  STRUCT
   STAT0 : ARRAY  [0 .. 255 ] OF //Temporary placeholder variable
   WORD  := W#16#0;
  END_STRUCT ;
BEGIN
   STAT0[0] := W#16#0;
   STAT0[1] := W#16#0;
   STAT0[2] := W#16#0;
   STAT0[3] := W#16#0;
   STAT0[4] := W#16#0;
   STAT0[5] := W#16#0;
   STAT0[6] := W#16#0;
   STAT0[7] := W#16#0;
   STAT0[8] := W#16#0;
   STAT0[9] := W#16#0;
   STAT0[10] := W#16#0;
   STAT0[11] := W#16#0;
   STAT0[12] := W#16#0;
   STAT0[13] := W#16#0;
   STAT0[14] := W#16#0;
   STAT0[15] := W#16#0;
   STAT0[16] := W#16#0;
   STAT0[17] := W#16#0;
   STAT0[18] := W#16#0;
   STAT0[19] := W#16#0;
   STAT0[20] := W#16#0;
   STAT0[21] := W#16#0;
   STAT0[22] := W#16#0;
   STAT0[23] := W#16#0;
   STAT0[24] := W#16#0;
   STAT0[25] := W#16#0;
   STAT0[26] := W#16#0;
   STAT0[27] := W#16#0;
   STAT0[28] := W#16#0;
   STAT0[29] := W#16#0;
   STAT0[30] := W#16#0;
   STAT0[31] := W#16#0;
   STAT0[32] := W#16#0;
   STAT0[33] := W#16#0;
   STAT0[34] := W#16#0;
   STAT0[35] := W#16#0;
   STAT0[36] := W#16#0;
   STAT0[37] := W#16#0;
   STAT0[38] := W#16#0;
   STAT0[39] := W#16#0;
   STAT0[40] := W#16#0;
   STAT0[41] := W#16#0;
   STAT0[42] := W#16#0;
   STAT0[43] := W#16#0;
   STAT0[44] := W#16#0;
   STAT0[45] := W#16#0;
   STAT0[46] := W#16#0;
   STAT0[47] := W#16#0;
   STAT0[48] := W#16#0;
   STAT0[49] := W#16#0;
   STAT0[50] := W#16#0;
   STAT0[51] := W#16#0;
   STAT0[52] := W#16#0;
   STAT0[53] := W#16#0;
   STAT0[54] := W#16#0;
   STAT0[55] := W#16#0;
   STAT0[56] := W#16#0;
   STAT0[57] := W#16#0;
   STAT0[58] := W#16#0;
   STAT0[59] := W#16#0;
   STAT0[60] := W#16#0;
   STAT0[61] := W#16#0;
   STAT0[62] := W#16#0;
   STAT0[63] := W#16#0;
   STAT0[64] := W#16#0;
   STAT0[65] := W#16#0;
   STAT0[66] := W#16#0;
   STAT0[67] := W#16#0;
   STAT0[68] := W#16#0;
   STAT0[69] := W#16#0;
   STAT0[70] := W#16#0;
   STAT0[71] := W#16#0;
   STAT0[72] := W#16#0;
   STAT0[73] := W#16#0;
   STAT0[74] := W#16#0;
   STAT0[75] := W#16#0;
   STAT0[76] := W#16#0;
   STAT0[77] := W#16#0;
   STAT0[78] := W#16#0;
   STAT0[79] := W#16#0;
   STAT0[80] := W#16#0;
   STAT0[81] := W#16#0;
   STAT0[82] := W#16#0;
   STAT0[83] := W#16#0;
   STAT0[84] := W#16#0;
   STAT0[85] := W#16#0;
   STAT0[86] := W#16#0;
   STAT0[87] := W#16#0;
   STAT0[88] := W#16#0;
   STAT0[89] := W#16#0;
   STAT0[90] := W#16#0;
   STAT0[91] := W#16#0;
   STAT0[92] := W#16#0;
   STAT0[93] := W#16#0;
   STAT0[94] := W#16#0;
   STAT0[95] := W#16#0;
   STAT0[96] := W#16#0;
   STAT0[97] := W#16#0;
   STAT0[98] := W#16#0;
   STAT0[99] := W#16#0;
   STAT0[100] := W#16#0;
   STAT0[101] := W#16#0;
   STAT0[102] := W#16#0;
   STAT0[103] := W#16#0;
   STAT0[104] := W#16#0;
   STAT0[105] := W#16#0;
   STAT0[106] := W#16#0;
   STAT0[107] := W#16#0;
   STAT0[108] := W#16#0;
   STAT0[109] := W#16#0;
   STAT0[110] := W#16#0;
   STAT0[111] := W#16#0;
   STAT0[112] := W#16#0;
   STAT0[113] := W#16#0;
   STAT0[114] := W#16#0;
   STAT0[115] := W#16#0;
   STAT0[116] := W#16#0;
   STAT0[117] := W#16#0;
   STAT0[118] := W#16#0;
   STAT0[119] := W#16#0;
   STAT0[120] := W#16#0;
   STAT0[121] := W#16#0;
   STAT0[122] := W#16#0;
   STAT0[123] := W#16#0;
   STAT0[124] := W#16#0;
   STAT0[125] := W#16#0;
   STAT0[126] := W#16#0;
   STAT0[127] := W#16#0;
   STAT0[128] := W#16#0;
   STAT0[129] := W#16#0;
   STAT0[130] := W#16#0;
   STAT0[131] := W#16#0;
   STAT0[132] := W#16#0;
   STAT0[133] := W#16#0;
   STAT0[134] := W#16#0;
   STAT0[135] := W#16#0;
   STAT0[136] := W#16#0;
   STAT0[137] := W#16#0;
   STAT0[138] := W#16#0;
   STAT0[139] := W#16#0;
   STAT0[140] := W#16#0;
   STAT0[141] := W#16#0;
   STAT0[142] := W#16#0;
   STAT0[143] := W#16#0;
   STAT0[144] := W#16#0;
   STAT0[145] := W#16#0;
   STAT0[146] := W#16#0;
   STAT0[147] := W#16#0;
   STAT0[148] := W#16#0;
   STAT0[149] := W#16#0;
   STAT0[150] := W#16#0;
   STAT0[151] := W#16#0;
   STAT0[152] := W#16#0;
   STAT0[153] := W#16#0;
   STAT0[154] := W#16#0;
   STAT0[155] := W#16#0;
   STAT0[156] := W#16#0;
   STAT0[157] := W#16#0;
   STAT0[158] := W#16#0;
   STAT0[159] := W#16#0;
   STAT0[160] := W#16#0;
   STAT0[161] := W#16#0;
   STAT0[162] := W#16#0;
   STAT0[163] := W#16#0;
   STAT0[164] := W#16#0;
   STAT0[165] := W#16#0;
   STAT0[166] := W#16#0;
   STAT0[167] := W#16#0;
   STAT0[168] := W#16#0;
   STAT0[169] := W#16#0;
   STAT0[170] := W#16#0;
   STAT0[171] := W#16#0;
   STAT0[172] := W#16#0;
   STAT0[173] := W#16#0;
   STAT0[174] := W#16#0;
   STAT0[175] := W#16#0;
   STAT0[176] := W#16#0;
   STAT0[177] := W#16#0;
   STAT0[178] := W#16#0;
   STAT0[179] := W#16#0;
   STAT0[180] := W#16#0;
   STAT0[181] := W#16#0;
   STAT0[182] := W#16#0;
   STAT0[183] := W#16#0;
   STAT0[184] := W#16#0;
   STAT0[185] := W#16#0;
   STAT0[186] := W#16#0;
   STAT0[187] := W#16#0;
   STAT0[188] := W#16#0;
   STAT0[189] := W#16#0;
   STAT0[190] := W#16#0;
   STAT0[191] := W#16#0;
   STAT0[192] := W#16#0;
   STAT0[193] := W#16#0;
   STAT0[194] := W#16#0;
   STAT0[195] := W#16#0;
   STAT0[196] := W#16#0;
   STAT0[197] := W#16#0;
   STAT0[198] := W#16#0;
   STAT0[199] := W#16#0;
   STAT0[200] := W#16#0;
   STAT0[201] := W#16#0;
   STAT0[202] := W#16#0;
   STAT0[203] := W#16#0;
   STAT0[204] := W#16#0;
   STAT0[205] := W#16#0;
   STAT0[206] := W#16#0;
   STAT0[207] := W#16#0;
   STAT0[208] := W#16#0;
   STAT0[209] := W#16#0;
   STAT0[210] := W#16#0;
   STAT0[211] := W#16#0;
   STAT0[212] := W#16#0;
   STAT0[213] := W#16#0;
   STAT0[214] := W#16#0;
   STAT0[215] := W#16#0;
   STAT0[216] := W#16#0;
   STAT0[217] := W#16#0;
   STAT0[218] := W#16#0;
   STAT0[219] := W#16#0;
   STAT0[220] := W#16#0;
   STAT0[221] := W#16#0;
   STAT0[222] := W#16#0;
   STAT0[223] := W#16#0;
   STAT0[224] := W#16#0;
   STAT0[225] := W#16#0;
   STAT0[226] := W#16#0;
   STAT0[227] := W#16#0;
   STAT0[228] := W#16#0;
   STAT0[229] := W#16#0;
   STAT0[230] := W#16#0;
   STAT0[231] := W#16#0;
   STAT0[232] := W#16#0;
   STAT0[233] := W#16#0;
   STAT0[234] := W#16#0;
   STAT0[235] := W#16#0;
   STAT0[236] := W#16#0;
   STAT0[237] := W#16#0;
   STAT0[238] := W#16#0;
   STAT0[239] := W#16#0;
   STAT0[240] := W#16#0;
   STAT0[241] := W#16#0;
   STAT0[242] := W#16#0;
   STAT0[243] := W#16#0;
   STAT0[244] := W#16#0;
   STAT0[245] := W#16#0;
   STAT0[246] := W#16#0;
   STAT0[247] := W#16#0;
   STAT0[248] := W#16#0;
   STAT0[249] := W#16#0;
   STAT0[250] := W#16#0;
   STAT0[251] := W#16#0;
   STAT0[252] := W#16#0;
   STAT0[253] := W#16#0;
   STAT0[254] := W#16#0;
   STAT0[255] := W#16#0;
END_DATA_BLOCK

DATA_BLOCK DB 325
TITLE =
VERSION : 0.1


  STRUCT
   DP_DIAG1 : ARRAY  [1 .. 100 ] OF BYTE ;
   DP_DIAG2 : ARRAY  [1 .. 100 ] OF BYTE ;
   DP_DIAG3 : ARRAY  [1 .. 100 ] OF BYTE ;
   DP_DIAG4 : ARRAY  [1 .. 100 ] OF BYTE ;
   DP_DIAG5 : ARRAY  [1 .. 100 ] OF BYTE ;
   DP_DIAG6 : ARRAY  [1 .. 100 ] OF BYTE ;
   DP_DIAG7 : ARRAY  [1 .. 100 ] OF BYTE ;
   DP_DIAG8 : ARRAY  [1 .. 100 ] OF BYTE ;
   DP_DIAG9 : ARRAY  [1 .. 100 ] OF BYTE ;
   DP_DIAG10 : ARRAY  [1 .. 100 ] OF BYTE ;
  END_STRUCT ;
BEGIN
   DP_DIAG1[1] := B#16#0;
   DP_DIAG1[2] := B#16#0;
   DP_DIAG1[3] := B#16#0;
   DP_DIAG1[4] := B#16#0;
   DP_DIAG1[5] := B#16#0;
   DP_DIAG1[6] := B#16#0;
   DP_DIAG1[7] := B#16#0;
   DP_DIAG1[8] := B#16#0;
   DP_DIAG1[9] := B#16#0;
   DP_DIAG1[10] := B#16#0;
   DP_DIAG1[11] := B#16#0;
   DP_DIAG1[12] := B#16#0;
   DP_DIAG1[13] := B#16#0;
   DP_DIAG1[14] := B#16#0;
   DP_DIAG1[15] := B#16#0;
   DP_DIAG1[16] := B#16#0;
   DP_DIAG1[17] := B#16#0;
   DP_DIAG1[18] := B#16#0;
   DP_DIAG1[19] := B#16#0;
   DP_DIAG1[20] := B#16#0;
   DP_DIAG1[21] := B#16#0;
   DP_DIAG1[22] := B#16#0;
   DP_DIAG1[23] := B#16#0;
   DP_DIAG1[24] := B#16#0;
   DP_DIAG1[25] := B#16#0;
   DP_DIAG1[26] := B#16#0;
   DP_DIAG1[27] := B#16#0;
   DP_DIAG1[28] := B#16#0;
   DP_DIAG1[29] := B#16#0;
   DP_DIAG1[30] := B#16#0;
   DP_DIAG1[31] := B#16#0;
   DP_DIAG1[32] := B#16#0;
   DP_DIAG1[33] := B#16#0;
   DP_DIAG1[34] := B#16#0;
   DP_DIAG1[35] := B#16#0;
   DP_DIAG1[36] := B#16#0;
   DP_DIAG1[37] := B#16#0;
   DP_DIAG1[38] := B#16#0;
   DP_DIAG1[39] := B#16#0;
   DP_DIAG1[40] := B#16#0;
   DP_DIAG1[41] := B#16#0;
   DP_DIAG1[42] := B#16#0;
   DP_DIAG1[43] := B#16#0;
   DP_DIAG1[44] := B#16#0;
   DP_DIAG1[45] := B#16#0;
   DP_DIAG1[46] := B#16#0;
   DP_DIAG1[47] := B#16#0;
   DP_DIAG1[48] := B#16#0;
   DP_DIAG1[49] := B#16#0;
   DP_DIAG1[50] := B#16#0;
   DP_DIAG1[51] := B#16#0;
   DP_DIAG1[52] := B#16#0;
   DP_DIAG1[53] := B#16#0;
   DP_DIAG1[54] := B#16#0;
   DP_DIAG1[55] := B#16#0;
   DP_DIAG1[56] := B#16#0;
   DP_DIAG1[57] := B#16#0;
   DP_DIAG1[58] := B#16#0;
   DP_DIAG1[59] := B#16#0;
   DP_DIAG1[60] := B#16#0;
   DP_DIAG1[61] := B#16#0;
   DP_DIAG1[62] := B#16#0;
   DP_DIAG1[63] := B#16#0;
   DP_DIAG1[64] := B#16#0;
   DP_DIAG1[65] := B#16#0;
   DP_DIAG1[66] := B#16#0;
   DP_DIAG1[67] := B#16#0;
   DP_DIAG1[68] := B#16#0;
   DP_DIAG1[69] := B#16#0;
   DP_DIAG1[70] := B#16#0;
   DP_DIAG1[71] := B#16#0;
   DP_DIAG1[72] := B#16#0;
   DP_DIAG1[73] := B#16#0;
   DP_DIAG1[74] := B#16#0;
   DP_DIAG1[75] := B#16#0;
   DP_DIAG1[76] := B#16#0;
   DP_DIAG1[77] := B#16#0;
   DP_DIAG1[78] := B#16#0;
   DP_DIAG1[79] := B#16#0;
   DP_DIAG1[80] := B#16#0;
   DP_DIAG1[81] := B#16#0;
   DP_DIAG1[82] := B#16#0;
   DP_DIAG1[83] := B#16#0;
   DP_DIAG1[84] := B#16#0;
   DP_DIAG1[85] := B#16#0;
   DP_DIAG1[86] := B#16#0;
   DP_DIAG1[87] := B#16#0;
   DP_DIAG1[88] := B#16#0;
   DP_DIAG1[89] := B#16#0;
   DP_DIAG1[90] := B#16#0;
   DP_DIAG1[91] := B#16#0;
   DP_DIAG1[92] := B#16#0;
   DP_DIAG1[93] := B#16#0;
   DP_DIAG1[94] := B#16#0;
   DP_DIAG1[95] := B#16#0;
   DP_DIAG1[96] := B#16#0;
   DP_DIAG1[97] := B#16#0;
   DP_DIAG1[98] := B#16#0;
   DP_DIAG1[99] := B#16#0;
   DP_DIAG1[100] := B#16#0;
   DP_DIAG2[1] := B#16#0;
   DP_DIAG2[2] := B#16#0;
   DP_DIAG2[3] := B#16#0;
   DP_DIAG2[4] := B#16#0;
   DP_DIAG2[5] := B#16#0;
   DP_DIAG2[6] := B#16#0;
   DP_DIAG2[7] := B#16#0;
   DP_DIAG2[8] := B#16#0;
   DP_DIAG2[9] := B#16#0;
   DP_DIAG2[10] := B#16#0;
   DP_DIAG2[11] := B#16#0;
   DP_DIAG2[12] := B#16#0;
   DP_DIAG2[13] := B#16#0;
   DP_DIAG2[14] := B#16#0;
   DP_DIAG2[15] := B#16#0;
   DP_DIAG2[16] := B#16#0;
   DP_DIAG2[17] := B#16#0;
   DP_DIAG2[18] := B#16#0;
   DP_DIAG2[19] := B#16#0;
   DP_DIAG2[20] := B#16#0;
   DP_DIAG2[21] := B#16#0;
   DP_DIAG2[22] := B#16#0;
   DP_DIAG2[23] := B#16#0;
   DP_DIAG2[24] := B#16#0;
   DP_DIAG2[25] := B#16#0;
   DP_DIAG2[26] := B#16#0;
   DP_DIAG2[27] := B#16#0;
   DP_DIAG2[28] := B#16#0;
   DP_DIAG2[29] := B#16#0;
   DP_DIAG2[30] := B#16#0;
   DP_DIAG2[31] := B#16#0;
   DP_DIAG2[32] := B#16#0;
   DP_DIAG2[33] := B#16#0;
   DP_DIAG2[34] := B#16#0;
   DP_DIAG2[35] := B#16#0;
   DP_DIAG2[36] := B#16#0;
   DP_DIAG2[37] := B#16#0;
   DP_DIAG2[38] := B#16#0;
   DP_DIAG2[39] := B#16#0;
   DP_DIAG2[40] := B#16#0;
   DP_DIAG2[41] := B#16#0;
   DP_DIAG2[42] := B#16#0;
   DP_DIAG2[43] := B#16#0;
   DP_DIAG2[44] := B#16#0;
   DP_DIAG2[45] := B#16#0;
   DP_DIAG2[46] := B#16#0;
   DP_DIAG2[47] := B#16#0;
   DP_DIAG2[48] := B#16#0;
   DP_DIAG2[49] := B#16#0;
   DP_DIAG2[50] := B#16#0;
   DP_DIAG2[51] := B#16#0;
   DP_DIAG2[52] := B#16#0;
   DP_DIAG2[53] := B#16#0;
   DP_DIAG2[54] := B#16#0;
   DP_DIAG2[55] := B#16#0;
   DP_DIAG2[56] := B#16#0;
   DP_DIAG2[57] := B#16#0;
   DP_DIAG2[58] := B#16#0;
   DP_DIAG2[59] := B#16#0;
   DP_DIAG2[60] := B#16#0;
   DP_DIAG2[61] := B#16#0;
   DP_DIAG2[62] := B#16#0;
   DP_DIAG2[63] := B#16#0;
   DP_DIAG2[64] := B#16#0;
   DP_DIAG2[65] := B#16#0;
   DP_DIAG2[66] := B#16#0;
   DP_DIAG2[67] := B#16#0;
   DP_DIAG2[68] := B#16#0;
   DP_DIAG2[69] := B#16#0;
   DP_DIAG2[70] := B#16#0;
   DP_DIAG2[71] := B#16#0;
   DP_DIAG2[72] := B#16#0;
   DP_DIAG2[73] := B#16#0;
   DP_DIAG2[74] := B#16#0;
   DP_DIAG2[75] := B#16#0;
   DP_DIAG2[76] := B#16#0;
   DP_DIAG2[77] := B#16#0;
   DP_DIAG2[78] := B#16#0;
   DP_DIAG2[79] := B#16#0;
   DP_DIAG2[80] := B#16#0;
   DP_DIAG2[81] := B#16#0;
   DP_DIAG2[82] := B#16#0;
   DP_DIAG2[83] := B#16#0;
   DP_DIAG2[84] := B#16#0;
   DP_DIAG2[85] := B#16#0;
   DP_DIAG2[86] := B#16#0;
   DP_DIAG2[87] := B#16#0;
   DP_DIAG2[88] := B#16#0;
   DP_DIAG2[89] := B#16#0;
   DP_DIAG2[90] := B#16#0;
   DP_DIAG2[91] := B#16#0;
   DP_DIAG2[92] := B#16#0;
   DP_DIAG2[93] := B#16#0;
   DP_DIAG2[94] := B#16#0;
   DP_DIAG2[95] := B#16#0;
   DP_DIAG2[96] := B#16#0;
   DP_DIAG2[97] := B#16#0;
   DP_DIAG2[98] := B#16#0;
   DP_DIAG2[99] := B#16#0;
   DP_DIAG2[100] := B#16#0;
   DP_DIAG3[1] := B#16#0;
   DP_DIAG3[2] := B#16#0;
   DP_DIAG3[3] := B#16#0;
   DP_DIAG3[4] := B#16#0;
   DP_DIAG3[5] := B#16#0;
   DP_DIAG3[6] := B#16#0;
   DP_DIAG3[7] := B#16#0;
   DP_DIAG3[8] := B#16#0;
   DP_DIAG3[9] := B#16#0;
   DP_DIAG3[10] := B#16#0;
   DP_DIAG3[11] := B#16#0;
   DP_DIAG3[12] := B#16#0;
   DP_DIAG3[13] := B#16#0;
   DP_DIAG3[14] := B#16#0;
   DP_DIAG3[15] := B#16#0;
   DP_DIAG3[16] := B#16#0;
   DP_DIAG3[17] := B#16#0;
   DP_DIAG3[18] := B#16#0;
   DP_DIAG3[19] := B#16#0;
   DP_DIAG3[20] := B#16#0;
   DP_DIAG3[21] := B#16#0;
   DP_DIAG3[22] := B#16#0;
   DP_DIAG3[23] := B#16#0;
   DP_DIAG3[24] := B#16#0;
   DP_DIAG3[25] := B#16#0;
   DP_DIAG3[26] := B#16#0;
   DP_DIAG3[27] := B#16#0;
   DP_DIAG3[28] := B#16#0;
   DP_DIAG3[29] := B#16#0;
   DP_DIAG3[30] := B#16#0;
   DP_DIAG3[31] := B#16#0;
   DP_DIAG3[32] := B#16#0;
   DP_DIAG3[33] := B#16#0;
   DP_DIAG3[34] := B#16#0;
   DP_DIAG3[35] := B#16#0;
   DP_DIAG3[36] := B#16#0;
   DP_DIAG3[37] := B#16#0;
   DP_DIAG3[38] := B#16#0;
   DP_DIAG3[39] := B#16#0;
   DP_DIAG3[40] := B#16#0;
   DP_DIAG3[41] := B#16#0;
   DP_DIAG3[42] := B#16#0;
   DP_DIAG3[43] := B#16#0;
   DP_DIAG3[44] := B#16#0;
   DP_DIAG3[45] := B#16#0;
   DP_DIAG3[46] := B#16#0;
   DP_DIAG3[47] := B#16#0;
   DP_DIAG3[48] := B#16#0;
   DP_DIAG3[49] := B#16#0;
   DP_DIAG3[50] := B#16#0;
   DP_DIAG3[51] := B#16#0;
   DP_DIAG3[52] := B#16#0;
   DP_DIAG3[53] := B#16#0;
   DP_DIAG3[54] := B#16#0;
   DP_DIAG3[55] := B#16#0;
   DP_DIAG3[56] := B#16#0;
   DP_DIAG3[57] := B#16#0;
   DP_DIAG3[58] := B#16#0;
   DP_DIAG3[59] := B#16#0;
   DP_DIAG3[60] := B#16#0;
   DP_DIAG3[61] := B#16#0;
   DP_DIAG3[62] := B#16#0;
   DP_DIAG3[63] := B#16#0;
   DP_DIAG3[64] := B#16#0;
   DP_DIAG3[65] := B#16#0;
   DP_DIAG3[66] := B#16#0;
   DP_DIAG3[67] := B#16#0;
   DP_DIAG3[68] := B#16#0;
   DP_DIAG3[69] := B#16#0;
   DP_DIAG3[70] := B#16#0;
   DP_DIAG3[71] := B#16#0;
   DP_DIAG3[72] := B#16#0;
   DP_DIAG3[73] := B#16#0;
   DP_DIAG3[74] := B#16#0;
   DP_DIAG3[75] := B#16#0;
   DP_DIAG3[76] := B#16#0;
   DP_DIAG3[77] := B#16#0;
   DP_DIAG3[78] := B#16#0;
   DP_DIAG3[79] := B#16#0;
   DP_DIAG3[80] := B#16#0;
   DP_DIAG3[81] := B#16#0;
   DP_DIAG3[82] := B#16#0;
   DP_DIAG3[83] := B#16#0;
   DP_DIAG3[84] := B#16#0;
   DP_DIAG3[85] := B#16#0;
   DP_DIAG3[86] := B#16#0;
   DP_DIAG3[87] := B#16#0;
   DP_DIAG3[88] := B#16#0;
   DP_DIAG3[89] := B#16#0;
   DP_DIAG3[90] := B#16#0;
   DP_DIAG3[91] := B#16#0;
   DP_DIAG3[92] := B#16#0;
   DP_DIAG3[93] := B#16#0;
   DP_DIAG3[94] := B#16#0;
   DP_DIAG3[95] := B#16#0;
   DP_DIAG3[96] := B#16#0;
   DP_DIAG3[97] := B#16#0;
   DP_DIAG3[98] := B#16#0;
   DP_DIAG3[99] := B#16#0;
   DP_DIAG3[100] := B#16#0;
   DP_DIAG4[1] := B#16#0;
   DP_DIAG4[2] := B#16#0;
   DP_DIAG4[3] := B#16#0;
   DP_DIAG4[4] := B#16#0;
   DP_DIAG4[5] := B#16#0;
   DP_DIAG4[6] := B#16#0;
   DP_DIAG4[7] := B#16#0;
   DP_DIAG4[8] := B#16#0;
   DP_DIAG4[9] := B#16#0;
   DP_DIAG4[10] := B#16#0;
   DP_DIAG4[11] := B#16#0;
   DP_DIAG4[12] := B#16#0;
   DP_DIAG4[13] := B#16#0;
   DP_DIAG4[14] := B#16#0;
   DP_DIAG4[15] := B#16#0;
   DP_DIAG4[16] := B#16#0;
   DP_DIAG4[17] := B#16#0;
   DP_DIAG4[18] := B#16#0;
   DP_DIAG4[19] := B#16#0;
   DP_DIAG4[20] := B#16#0;
   DP_DIAG4[21] := B#16#0;
   DP_DIAG4[22] := B#16#0;
   DP_DIAG4[23] := B#16#0;
   DP_DIAG4[24] := B#16#0;
   DP_DIAG4[25] := B#16#0;
   DP_DIAG4[26] := B#16#0;
   DP_DIAG4[27] := B#16#0;
   DP_DIAG4[28] := B#16#0;
   DP_DIAG4[29] := B#16#0;
   DP_DIAG4[30] := B#16#0;
   DP_DIAG4[31] := B#16#0;
   DP_DIAG4[32] := B#16#0;
   DP_DIAG4[33] := B#16#0;
   DP_DIAG4[34] := B#16#0;
   DP_DIAG4[35] := B#16#0;
   DP_DIAG4[36] := B#16#0;
   DP_DIAG4[37] := B#16#0;
   DP_DIAG4[38] := B#16#0;
   DP_DIAG4[39] := B#16#0;
   DP_DIAG4[40] := B#16#0;
   DP_DIAG4[41] := B#16#0;
   DP_DIAG4[42] := B#16#0;
   DP_DIAG4[43] := B#16#0;
   DP_DIAG4[44] := B#16#0;
   DP_DIAG4[45] := B#16#0;
   DP_DIAG4[46] := B#16#0;
   DP_DIAG4[47] := B#16#0;
   DP_DIAG4[48] := B#16#0;
   DP_DIAG4[49] := B#16#0;
   DP_DIAG4[50] := B#16#0;
   DP_DIAG4[51] := B#16#0;
   DP_DIAG4[52] := B#16#0;
   DP_DIAG4[53] := B#16#0;
   DP_DIAG4[54] := B#16#0;
   DP_DIAG4[55] := B#16#0;
   DP_DIAG4[56] := B#16#0;
   DP_DIAG4[57] := B#16#0;
   DP_DIAG4[58] := B#16#0;
   DP_DIAG4[59] := B#16#0;
   DP_DIAG4[60] := B#16#0;
   DP_DIAG4[61] := B#16#0;
   DP_DIAG4[62] := B#16#0;
   DP_DIAG4[63] := B#16#0;
   DP_DIAG4[64] := B#16#0;
   DP_DIAG4[65] := B#16#0;
   DP_DIAG4[66] := B#16#0;
   DP_DIAG4[67] := B#16#0;
   DP_DIAG4[68] := B#16#0;
   DP_DIAG4[69] := B#16#0;
   DP_DIAG4[70] := B#16#0;
   DP_DIAG4[71] := B#16#0;
   DP_DIAG4[72] := B#16#0;
   DP_DIAG4[73] := B#16#0;
   DP_DIAG4[74] := B#16#0;
   DP_DIAG4[75] := B#16#0;
   DP_DIAG4[76] := B#16#0;
   DP_DIAG4[77] := B#16#0;
   DP_DIAG4[78] := B#16#0;
   DP_DIAG4[79] := B#16#0;
   DP_DIAG4[80] := B#16#0;
   DP_DIAG4[81] := B#16#0;
   DP_DIAG4[82] := B#16#0;
   DP_DIAG4[83] := B#16#0;
   DP_DIAG4[84] := B#16#0;
   DP_DIAG4[85] := B#16#0;
   DP_DIAG4[86] := B#16#0;
   DP_DIAG4[87] := B#16#0;
   DP_DIAG4[88] := B#16#0;
   DP_DIAG4[89] := B#16#0;
   DP_DIAG4[90] := B#16#0;
   DP_DIAG4[91] := B#16#0;
   DP_DIAG4[92] := B#16#0;
   DP_DIAG4[93] := B#16#0;
   DP_DIAG4[94] := B#16#0;
   DP_DIAG4[95] := B#16#0;
   DP_DIAG4[96] := B#16#0;
   DP_DIAG4[97] := B#16#0;
   DP_DIAG4[98] := B#16#0;
   DP_DIAG4[99] := B#16#0;
   DP_DIAG4[100] := B#16#0;
   DP_DIAG5[1] := B#16#0;
   DP_DIAG5[2] := B#16#0;
   DP_DIAG5[3] := B#16#0;
   DP_DIAG5[4] := B#16#0;
   DP_DIAG5[5] := B#16#0;
   DP_DIAG5[6] := B#16#0;
   DP_DIAG5[7] := B#16#0;
   DP_DIAG5[8] := B#16#0;
   DP_DIAG5[9] := B#16#0;
   DP_DIAG5[10] := B#16#0;
   DP_DIAG5[11] := B#16#0;
   DP_DIAG5[12] := B#16#0;
   DP_DIAG5[13] := B#16#0;
   DP_DIAG5[14] := B#16#0;
   DP_DIAG5[15] := B#16#0;
   DP_DIAG5[16] := B#16#0;
   DP_DIAG5[17] := B#16#0;
   DP_DIAG5[18] := B#16#0;
   DP_DIAG5[19] := B#16#0;
   DP_DIAG5[20] := B#16#0;
   DP_DIAG5[21] := B#16#0;
   DP_DIAG5[22] := B#16#0;
   DP_DIAG5[23] := B#16#0;
   DP_DIAG5[24] := B#16#0;
   DP_DIAG5[25] := B#16#0;
   DP_DIAG5[26] := B#16#0;
   DP_DIAG5[27] := B#16#0;
   DP_DIAG5[28] := B#16#0;
   DP_DIAG5[29] := B#16#0;
   DP_DIAG5[30] := B#16#0;
   DP_DIAG5[31] := B#16#0;
   DP_DIAG5[32] := B#16#0;
   DP_DIAG5[33] := B#16#0;
   DP_DIAG5[34] := B#16#0;
   DP_DIAG5[35] := B#16#0;
   DP_DIAG5[36] := B#16#0;
   DP_DIAG5[37] := B#16#0;
   DP_DIAG5[38] := B#16#0;
   DP_DIAG5[39] := B#16#0;
   DP_DIAG5[40] := B#16#0;
   DP_DIAG5[41] := B#16#0;
   DP_DIAG5[42] := B#16#0;
   DP_DIAG5[43] := B#16#0;
   DP_DIAG5[44] := B#16#0;
   DP_DIAG5[45] := B#16#0;
   DP_DIAG5[46] := B#16#0;
   DP_DIAG5[47] := B#16#0;
   DP_DIAG5[48] := B#16#0;
   DP_DIAG5[49] := B#16#0;
   DP_DIAG5[50] := B#16#0;
   DP_DIAG5[51] := B#16#0;
   DP_DIAG5[52] := B#16#0;
   DP_DIAG5[53] := B#16#0;
   DP_DIAG5[54] := B#16#0;
   DP_DIAG5[55] := B#16#0;
   DP_DIAG5[56] := B#16#0;
   DP_DIAG5[57] := B#16#0;
   DP_DIAG5[58] := B#16#0;
   DP_DIAG5[59] := B#16#0;
   DP_DIAG5[60] := B#16#0;
   DP_DIAG5[61] := B#16#0;
   DP_DIAG5[62] := B#16#0;
   DP_DIAG5[63] := B#16#0;
   DP_DIAG5[64] := B#16#0;
   DP_DIAG5[65] := B#16#0;
   DP_DIAG5[66] := B#16#0;
   DP_DIAG5[67] := B#16#0;
   DP_DIAG5[68] := B#16#0;
   DP_DIAG5[69] := B#16#0;
   DP_DIAG5[70] := B#16#0;
   DP_DIAG5[71] := B#16#0;
   DP_DIAG5[72] := B#16#0;
   DP_DIAG5[73] := B#16#0;
   DP_DIAG5[74] := B#16#0;
   DP_DIAG5[75] := B#16#0;
   DP_DIAG5[76] := B#16#0;
   DP_DIAG5[77] := B#16#0;
   DP_DIAG5[78] := B#16#0;
   DP_DIAG5[79] := B#16#0;
   DP_DIAG5[80] := B#16#0;
   DP_DIAG5[81] := B#16#0;
   DP_DIAG5[82] := B#16#0;
   DP_DIAG5[83] := B#16#0;
   DP_DIAG5[84] := B#16#0;
   DP_DIAG5[85] := B#16#0;
   DP_DIAG5[86] := B#16#0;
   DP_DIAG5[87] := B#16#0;
   DP_DIAG5[88] := B#16#0;
   DP_DIAG5[89] := B#16#0;
   DP_DIAG5[90] := B#16#0;
   DP_DIAG5[91] := B#16#0;
   DP_DIAG5[92] := B#16#0;
   DP_DIAG5[93] := B#16#0;
   DP_DIAG5[94] := B#16#0;
   DP_DIAG5[95] := B#16#0;
   DP_DIAG5[96] := B#16#0;
   DP_DIAG5[97] := B#16#0;
   DP_DIAG5[98] := B#16#0;
   DP_DIAG5[99] := B#16#0;
   DP_DIAG5[100] := B#16#0;
   DP_DIAG6[1] := B#16#0;
   DP_DIAG6[2] := B#16#0;
   DP_DIAG6[3] := B#16#0;
   DP_DIAG6[4] := B#16#0;
   DP_DIAG6[5] := B#16#0;
   DP_DIAG6[6] := B#16#0;
   DP_DIAG6[7] := B#16#0;
   DP_DIAG6[8] := B#16#0;
   DP_DIAG6[9] := B#16#0;
   DP_DIAG6[10] := B#16#0;
   DP_DIAG6[11] := B#16#0;
   DP_DIAG6[12] := B#16#0;
   DP_DIAG6[13] := B#16#0;
   DP_DIAG6[14] := B#16#0;
   DP_DIAG6[15] := B#16#0;
   DP_DIAG6[16] := B#16#0;
   DP_DIAG6[17] := B#16#0;
   DP_DIAG6[18] := B#16#0;
   DP_DIAG6[19] := B#16#0;
   DP_DIAG6[20] := B#16#0;
   DP_DIAG6[21] := B#16#0;
   DP_DIAG6[22] := B#16#0;
   DP_DIAG6[23] := B#16#0;
   DP_DIAG6[24] := B#16#0;
   DP_DIAG6[25] := B#16#0;
   DP_DIAG6[26] := B#16#0;
   DP_DIAG6[27] := B#16#0;
   DP_DIAG6[28] := B#16#0;
   DP_DIAG6[29] := B#16#0;
   DP_DIAG6[30] := B#16#0;
   DP_DIAG6[31] := B#16#0;
   DP_DIAG6[32] := B#16#0;
   DP_DIAG6[33] := B#16#0;
   DP_DIAG6[34] := B#16#0;
   DP_DIAG6[35] := B#16#0;
   DP_DIAG6[36] := B#16#0;
   DP_DIAG6[37] := B#16#0;
   DP_DIAG6[38] := B#16#0;
   DP_DIAG6[39] := B#16#0;
   DP_DIAG6[40] := B#16#0;
   DP_DIAG6[41] := B#16#0;
   DP_DIAG6[42] := B#16#0;
   DP_DIAG6[43] := B#16#0;
   DP_DIAG6[44] := B#16#0;
   DP_DIAG6[45] := B#16#0;
   DP_DIAG6[46] := B#16#0;
   DP_DIAG6[47] := B#16#0;
   DP_DIAG6[48] := B#16#0;
   DP_DIAG6[49] := B#16#0;
   DP_DIAG6[50] := B#16#0;
   DP_DIAG6[51] := B#16#0;
   DP_DIAG6[52] := B#16#0;
   DP_DIAG6[53] := B#16#0;
   DP_DIAG6[54] := B#16#0;
   DP_DIAG6[55] := B#16#0;
   DP_DIAG6[56] := B#16#0;
   DP_DIAG6[57] := B#16#0;
   DP_DIAG6[58] := B#16#0;
   DP_DIAG6[59] := B#16#0;
   DP_DIAG6[60] := B#16#0;
   DP_DIAG6[61] := B#16#0;
   DP_DIAG6[62] := B#16#0;
   DP_DIAG6[63] := B#16#0;
   DP_DIAG6[64] := B#16#0;
   DP_DIAG6[65] := B#16#0;
   DP_DIAG6[66] := B#16#0;
   DP_DIAG6[67] := B#16#0;
   DP_DIAG6[68] := B#16#0;
   DP_DIAG6[69] := B#16#0;
   DP_DIAG6[70] := B#16#0;
   DP_DIAG6[71] := B#16#0;
   DP_DIAG6[72] := B#16#0;
   DP_DIAG6[73] := B#16#0;
   DP_DIAG6[74] := B#16#0;
   DP_DIAG6[75] := B#16#0;
   DP_DIAG6[76] := B#16#0;
   DP_DIAG6[77] := B#16#0;
   DP_DIAG6[78] := B#16#0;
   DP_DIAG6[79] := B#16#0;
   DP_DIAG6[80] := B#16#0;
   DP_DIAG6[81] := B#16#0;
   DP_DIAG6[82] := B#16#0;
   DP_DIAG6[83] := B#16#0;
   DP_DIAG6[84] := B#16#0;
   DP_DIAG6[85] := B#16#0;
   DP_DIAG6[86] := B#16#0;
   DP_DIAG6[87] := B#16#0;
   DP_DIAG6[88] := B#16#0;
   DP_DIAG6[89] := B#16#0;
   DP_DIAG6[90] := B#16#0;
   DP_DIAG6[91] := B#16#0;
   DP_DIAG6[92] := B#16#0;
   DP_DIAG6[93] := B#16#0;
   DP_DIAG6[94] := B#16#0;
   DP_DIAG6[95] := B#16#0;
   DP_DIAG6[96] := B#16#0;
   DP_DIAG6[97] := B#16#0;
   DP_DIAG6[98] := B#16#0;
   DP_DIAG6[99] := B#16#0;
   DP_DIAG6[100] := B#16#0;
   DP_DIAG7[1] := B#16#0;
   DP_DIAG7[2] := B#16#0;
   DP_DIAG7[3] := B#16#0;
   DP_DIAG7[4] := B#16#0;
   DP_DIAG7[5] := B#16#0;
   DP_DIAG7[6] := B#16#0;
   DP_DIAG7[7] := B#16#0;
   DP_DIAG7[8] := B#16#0;
   DP_DIAG7[9] := B#16#0;
   DP_DIAG7[10] := B#16#0;
   DP_DIAG7[11] := B#16#0;
   DP_DIAG7[12] := B#16#0;
   DP_DIAG7[13] := B#16#0;
   DP_DIAG7[14] := B#16#0;
   DP_DIAG7[15] := B#16#0;
   DP_DIAG7[16] := B#16#0;
   DP_DIAG7[17] := B#16#0;
   DP_DIAG7[18] := B#16#0;
   DP_DIAG7[19] := B#16#0;
   DP_DIAG7[20] := B#16#0;
   DP_DIAG7[21] := B#16#0;
   DP_DIAG7[22] := B#16#0;
   DP_DIAG7[23] := B#16#0;
   DP_DIAG7[24] := B#16#0;
   DP_DIAG7[25] := B#16#0;
   DP_DIAG7[26] := B#16#0;
   DP_DIAG7[27] := B#16#0;
   DP_DIAG7[28] := B#16#0;
   DP_DIAG7[29] := B#16#0;
   DP_DIAG7[30] := B#16#0;
   DP_DIAG7[31] := B#16#0;
   DP_DIAG7[32] := B#16#0;
   DP_DIAG7[33] := B#16#0;
   DP_DIAG7[34] := B#16#0;
   DP_DIAG7[35] := B#16#0;
   DP_DIAG7[36] := B#16#0;
   DP_DIAG7[37] := B#16#0;
   DP_DIAG7[38] := B#16#0;
   DP_DIAG7[39] := B#16#0;
   DP_DIAG7[40] := B#16#0;
   DP_DIAG7[41] := B#16#0;
   DP_DIAG7[42] := B#16#0;
   DP_DIAG7[43] := B#16#0;
   DP_DIAG7[44] := B#16#0;
   DP_DIAG7[45] := B#16#0;
   DP_DIAG7[46] := B#16#0;
   DP_DIAG7[47] := B#16#0;
   DP_DIAG7[48] := B#16#0;
   DP_DIAG7[49] := B#16#0;
   DP_DIAG7[50] := B#16#0;
   DP_DIAG7[51] := B#16#0;
   DP_DIAG7[52] := B#16#0;
   DP_DIAG7[53] := B#16#0;
   DP_DIAG7[54] := B#16#0;
   DP_DIAG7[55] := B#16#0;
   DP_DIAG7[56] := B#16#0;
   DP_DIAG7[57] := B#16#0;
   DP_DIAG7[58] := B#16#0;
   DP_DIAG7[59] := B#16#0;
   DP_DIAG7[60] := B#16#0;
   DP_DIAG7[61] := B#16#0;
   DP_DIAG7[62] := B#16#0;
   DP_DIAG7[63] := B#16#0;
   DP_DIAG7[64] := B#16#0;
   DP_DIAG7[65] := B#16#0;
   DP_DIAG7[66] := B#16#0;
   DP_DIAG7[67] := B#16#0;
   DP_DIAG7[68] := B#16#0;
   DP_DIAG7[69] := B#16#0;
   DP_DIAG7[70] := B#16#0;
   DP_DIAG7[71] := B#16#0;
   DP_DIAG7[72] := B#16#0;
   DP_DIAG7[73] := B#16#0;
   DP_DIAG7[74] := B#16#0;
   DP_DIAG7[75] := B#16#0;
   DP_DIAG7[76] := B#16#0;
   DP_DIAG7[77] := B#16#0;
   DP_DIAG7[78] := B#16#0;
   DP_DIAG7[79] := B#16#0;
   DP_DIAG7[80] := B#16#0;
   DP_DIAG7[81] := B#16#0;
   DP_DIAG7[82] := B#16#0;
   DP_DIAG7[83] := B#16#0;
   DP_DIAG7[84] := B#16#0;
   DP_DIAG7[85] := B#16#0;
   DP_DIAG7[86] := B#16#0;
   DP_DIAG7[87] := B#16#0;
   DP_DIAG7[88] := B#16#0;
   DP_DIAG7[89] := B#16#0;
   DP_DIAG7[90] := B#16#0;
   DP_DIAG7[91] := B#16#0;
   DP_DIAG7[92] := B#16#0;
   DP_DIAG7[93] := B#16#0;
   DP_DIAG7[94] := B#16#0;
   DP_DIAG7[95] := B#16#0;
   DP_DIAG7[96] := B#16#0;
   DP_DIAG7[97] := B#16#0;
   DP_DIAG7[98] := B#16#0;
   DP_DIAG7[99] := B#16#0;
   DP_DIAG7[100] := B#16#0;
   DP_DIAG8[1] := B#16#0;
   DP_DIAG8[2] := B#16#0;
   DP_DIAG8[3] := B#16#0;
   DP_DIAG8[4] := B#16#0;
   DP_DIAG8[5] := B#16#0;
   DP_DIAG8[6] := B#16#0;
   DP_DIAG8[7] := B#16#0;
   DP_DIAG8[8] := B#16#0;
   DP_DIAG8[9] := B#16#0;
   DP_DIAG8[10] := B#16#0;
   DP_DIAG8[11] := B#16#0;
   DP_DIAG8[12] := B#16#0;
   DP_DIAG8[13] := B#16#0;
   DP_DIAG8[14] := B#16#0;
   DP_DIAG8[15] := B#16#0;
   DP_DIAG8[16] := B#16#0;
   DP_DIAG8[17] := B#16#0;
   DP_DIAG8[18] := B#16#0;
   DP_DIAG8[19] := B#16#0;
   DP_DIAG8[20] := B#16#0;
   DP_DIAG8[21] := B#16#0;
   DP_DIAG8[22] := B#16#0;
   DP_DIAG8[23] := B#16#0;
   DP_DIAG8[24] := B#16#0;
   DP_DIAG8[25] := B#16#0;
   DP_DIAG8[26] := B#16#0;
   DP_DIAG8[27] := B#16#0;
   DP_DIAG8[28] := B#16#0;
   DP_DIAG8[29] := B#16#0;
   DP_DIAG8[30] := B#16#0;
   DP_DIAG8[31] := B#16#0;
   DP_DIAG8[32] := B#16#0;
   DP_DIAG8[33] := B#16#0;
   DP_DIAG8[34] := B#16#0;
   DP_DIAG8[35] := B#16#0;
   DP_DIAG8[36] := B#16#0;
   DP_DIAG8[37] := B#16#0;
   DP_DIAG8[38] := B#16#0;
   DP_DIAG8[39] := B#16#0;
   DP_DIAG8[40] := B#16#0;
   DP_DIAG8[41] := B#16#0;
   DP_DIAG8[42] := B#16#0;
   DP_DIAG8[43] := B#16#0;
   DP_DIAG8[44] := B#16#0;
   DP_DIAG8[45] := B#16#0;
   DP_DIAG8[46] := B#16#0;
   DP_DIAG8[47] := B#16#0;
   DP_DIAG8[48] := B#16#0;
   DP_DIAG8[49] := B#16#0;
   DP_DIAG8[50] := B#16#0;
   DP_DIAG8[51] := B#16#0;
   DP_DIAG8[52] := B#16#0;
   DP_DIAG8[53] := B#16#0;
   DP_DIAG8[54] := B#16#0;
   DP_DIAG8[55] := B#16#0;
   DP_DIAG8[56] := B#16#0;
   DP_DIAG8[57] := B#16#0;
   DP_DIAG8[58] := B#16#0;
   DP_DIAG8[59] := B#16#0;
   DP_DIAG8[60] := B#16#0;
   DP_DIAG8[61] := B#16#0;
   DP_DIAG8[62] := B#16#0;
   DP_DIAG8[63] := B#16#0;
   DP_DIAG8[64] := B#16#0;
   DP_DIAG8[65] := B#16#0;
   DP_DIAG8[66] := B#16#0;
   DP_DIAG8[67] := B#16#0;
   DP_DIAG8[68] := B#16#0;
   DP_DIAG8[69] := B#16#0;
   DP_DIAG8[70] := B#16#0;
   DP_DIAG8[71] := B#16#0;
   DP_DIAG8[72] := B#16#0;
   DP_DIAG8[73] := B#16#0;
   DP_DIAG8[74] := B#16#0;
   DP_DIAG8[75] := B#16#0;
   DP_DIAG8[76] := B#16#0;
   DP_DIAG8[77] := B#16#0;
   DP_DIAG8[78] := B#16#0;
   DP_DIAG8[79] := B#16#0;
   DP_DIAG8[80] := B#16#0;
   DP_DIAG8[81] := B#16#0;
   DP_DIAG8[82] := B#16#0;
   DP_DIAG8[83] := B#16#0;
   DP_DIAG8[84] := B#16#0;
   DP_DIAG8[85] := B#16#0;
   DP_DIAG8[86] := B#16#0;
   DP_DIAG8[87] := B#16#0;
   DP_DIAG8[88] := B#16#0;
   DP_DIAG8[89] := B#16#0;
   DP_DIAG8[90] := B#16#0;
   DP_DIAG8[91] := B#16#0;
   DP_DIAG8[92] := B#16#0;
   DP_DIAG8[93] := B#16#0;
   DP_DIAG8[94] := B#16#0;
   DP_DIAG8[95] := B#16#0;
   DP_DIAG8[96] := B#16#0;
   DP_DIAG8[97] := B#16#0;
   DP_DIAG8[98] := B#16#0;
   DP_DIAG8[99] := B#16#0;
   DP_DIAG8[100] := B#16#0;
   DP_DIAG9[1] := B#16#0;
   DP_DIAG9[2] := B#16#0;
   DP_DIAG9[3] := B#16#0;
   DP_DIAG9[4] := B#16#0;
   DP_DIAG9[5] := B#16#0;
   DP_DIAG9[6] := B#16#0;
   DP_DIAG9[7] := B#16#0;
   DP_DIAG9[8] := B#16#0;
   DP_DIAG9[9] := B#16#0;
   DP_DIAG9[10] := B#16#0;
   DP_DIAG9[11] := B#16#0;
   DP_DIAG9[12] := B#16#0;
   DP_DIAG9[13] := B#16#0;
   DP_DIAG9[14] := B#16#0;
   DP_DIAG9[15] := B#16#0;
   DP_DIAG9[16] := B#16#0;
   DP_DIAG9[17] := B#16#0;
   DP_DIAG9[18] := B#16#0;
   DP_DIAG9[19] := B#16#0;
   DP_DIAG9[20] := B#16#0;
   DP_DIAG9[21] := B#16#0;
   DP_DIAG9[22] := B#16#0;
   DP_DIAG9[23] := B#16#0;
   DP_DIAG9[24] := B#16#0;
   DP_DIAG9[25] := B#16#0;
   DP_DIAG9[26] := B#16#0;
   DP_DIAG9[27] := B#16#0;
   DP_DIAG9[28] := B#16#0;
   DP_DIAG9[29] := B#16#0;
   DP_DIAG9[30] := B#16#0;
   DP_DIAG9[31] := B#16#0;
   DP_DIAG9[32] := B#16#0;
   DP_DIAG9[33] := B#16#0;
   DP_DIAG9[34] := B#16#0;
   DP_DIAG9[35] := B#16#0;
   DP_DIAG9[36] := B#16#0;
   DP_DIAG9[37] := B#16#0;
   DP_DIAG9[38] := B#16#0;
   DP_DIAG9[39] := B#16#0;
   DP_DIAG9[40] := B#16#0;
   DP_DIAG9[41] := B#16#0;
   DP_DIAG9[42] := B#16#0;
   DP_DIAG9[43] := B#16#0;
   DP_DIAG9[44] := B#16#0;
   DP_DIAG9[45] := B#16#0;
   DP_DIAG9[46] := B#16#0;
   DP_DIAG9[47] := B#16#0;
   DP_DIAG9[48] := B#16#0;
   DP_DIAG9[49] := B#16#0;
   DP_DIAG9[50] := B#16#0;
   DP_DIAG9[51] := B#16#0;
   DP_DIAG9[52] := B#16#0;
   DP_DIAG9[53] := B#16#0;
   DP_DIAG9[54] := B#16#0;
   DP_DIAG9[55] := B#16#0;
   DP_DIAG9[56] := B#16#0;
   DP_DIAG9[57] := B#16#0;
   DP_DIAG9[58] := B#16#0;
   DP_DIAG9[59] := B#16#0;
   DP_DIAG9[60] := B#16#0;
   DP_DIAG9[61] := B#16#0;
   DP_DIAG9[62] := B#16#0;
   DP_DIAG9[63] := B#16#0;
   DP_DIAG9[64] := B#16#0;
   DP_DIAG9[65] := B#16#0;
   DP_DIAG9[66] := B#16#0;
   DP_DIAG9[67] := B#16#0;
   DP_DIAG9[68] := B#16#0;
   DP_DIAG9[69] := B#16#0;
   DP_DIAG9[70] := B#16#0;
   DP_DIAG9[71] := B#16#0;
   DP_DIAG9[72] := B#16#0;
   DP_DIAG9[73] := B#16#0;
   DP_DIAG9[74] := B#16#0;
   DP_DIAG9[75] := B#16#0;
   DP_DIAG9[76] := B#16#0;
   DP_DIAG9[77] := B#16#0;
   DP_DIAG9[78] := B#16#0;
   DP_DIAG9[79] := B#16#0;
   DP_DIAG9[80] := B#16#0;
   DP_DIAG9[81] := B#16#0;
   DP_DIAG9[82] := B#16#0;
   DP_DIAG9[83] := B#16#0;
   DP_DIAG9[84] := B#16#0;
   DP_DIAG9[85] := B#16#0;
   DP_DIAG9[86] := B#16#0;
   DP_DIAG9[87] := B#16#0;
   DP_DIAG9[88] := B#16#0;
   DP_DIAG9[89] := B#16#0;
   DP_DIAG9[90] := B#16#0;
   DP_DIAG9[91] := B#16#0;
   DP_DIAG9[92] := B#16#0;
   DP_DIAG9[93] := B#16#0;
   DP_DIAG9[94] := B#16#0;
   DP_DIAG9[95] := B#16#0;
   DP_DIAG9[96] := B#16#0;
   DP_DIAG9[97] := B#16#0;
   DP_DIAG9[98] := B#16#0;
   DP_DIAG9[99] := B#16#0;
   DP_DIAG9[100] := B#16#0;
   DP_DIAG10[1] := B#16#0;
   DP_DIAG10[2] := B#16#0;
   DP_DIAG10[3] := B#16#0;
   DP_DIAG10[4] := B#16#0;
   DP_DIAG10[5] := B#16#0;
   DP_DIAG10[6] := B#16#0;
   DP_DIAG10[7] := B#16#0;
   DP_DIAG10[8] := B#16#0;
   DP_DIAG10[9] := B#16#0;
   DP_DIAG10[10] := B#16#0;
   DP_DIAG10[11] := B#16#0;
   DP_DIAG10[12] := B#16#0;
   DP_DIAG10[13] := B#16#0;
   DP_DIAG10[14] := B#16#0;
   DP_DIAG10[15] := B#16#0;
   DP_DIAG10[16] := B#16#0;
   DP_DIAG10[17] := B#16#0;
   DP_DIAG10[18] := B#16#0;
   DP_DIAG10[19] := B#16#0;
   DP_DIAG10[20] := B#16#0;
   DP_DIAG10[21] := B#16#0;
   DP_DIAG10[22] := B#16#0;
   DP_DIAG10[23] := B#16#0;
   DP_DIAG10[24] := B#16#0;
   DP_DIAG10[25] := B#16#0;
   DP_DIAG10[26] := B#16#0;
   DP_DIAG10[27] := B#16#0;
   DP_DIAG10[28] := B#16#0;
   DP_DIAG10[29] := B#16#0;
   DP_DIAG10[30] := B#16#0;
   DP_DIAG10[31] := B#16#0;
   DP_DIAG10[32] := B#16#0;
   DP_DIAG10[33] := B#16#0;
   DP_DIAG10[34] := B#16#0;
   DP_DIAG10[35] := B#16#0;
   DP_DIAG10[36] := B#16#0;
   DP_DIAG10[37] := B#16#0;
   DP_DIAG10[38] := B#16#0;
   DP_DIAG10[39] := B#16#0;
   DP_DIAG10[40] := B#16#0;
   DP_DIAG10[41] := B#16#0;
   DP_DIAG10[42] := B#16#0;
   DP_DIAG10[43] := B#16#0;
   DP_DIAG10[44] := B#16#0;
   DP_DIAG10[45] := B#16#0;
   DP_DIAG10[46] := B#16#0;
   DP_DIAG10[47] := B#16#0;
   DP_DIAG10[48] := B#16#0;
   DP_DIAG10[49] := B#16#0;
   DP_DIAG10[50] := B#16#0;
   DP_DIAG10[51] := B#16#0;
   DP_DIAG10[52] := B#16#0;
   DP_DIAG10[53] := B#16#0;
   DP_DIAG10[54] := B#16#0;
   DP_DIAG10[55] := B#16#0;
   DP_DIAG10[56] := B#16#0;
   DP_DIAG10[57] := B#16#0;
   DP_DIAG10[58] := B#16#0;
   DP_DIAG10[59] := B#16#0;
   DP_DIAG10[60] := B#16#0;
   DP_DIAG10[61] := B#16#0;
   DP_DIAG10[62] := B#16#0;
   DP_DIAG10[63] := B#16#0;
   DP_DIAG10[64] := B#16#0;
   DP_DIAG10[65] := B#16#0;
   DP_DIAG10[66] := B#16#0;
   DP_DIAG10[67] := B#16#0;
   DP_DIAG10[68] := B#16#0;
   DP_DIAG10[69] := B#16#0;
   DP_DIAG10[70] := B#16#0;
   DP_DIAG10[71] := B#16#0;
   DP_DIAG10[72] := B#16#0;
   DP_DIAG10[73] := B#16#0;
   DP_DIAG10[74] := B#16#0;
   DP_DIAG10[75] := B#16#0;
   DP_DIAG10[76] := B#16#0;
   DP_DIAG10[77] := B#16#0;
   DP_DIAG10[78] := B#16#0;
   DP_DIAG10[79] := B#16#0;
   DP_DIAG10[80] := B#16#0;
   DP_DIAG10[81] := B#16#0;
   DP_DIAG10[82] := B#16#0;
   DP_DIAG10[83] := B#16#0;
   DP_DIAG10[84] := B#16#0;
   DP_DIAG10[85] := B#16#0;
   DP_DIAG10[86] := B#16#0;
   DP_DIAG10[87] := B#16#0;
   DP_DIAG10[88] := B#16#0;
   DP_DIAG10[89] := B#16#0;
   DP_DIAG10[90] := B#16#0;
   DP_DIAG10[91] := B#16#0;
   DP_DIAG10[92] := B#16#0;
   DP_DIAG10[93] := B#16#0;
   DP_DIAG10[94] := B#16#0;
   DP_DIAG10[95] := B#16#0;
   DP_DIAG10[96] := B#16#0;
   DP_DIAG10[97] := B#16#0;
   DP_DIAG10[98] := B#16#0;
   DP_DIAG10[99] := B#16#0;
   DP_DIAG10[100] := B#16#0;
END_DATA_BLOCK

FUNCTION_BLOCK FB 402
TITLE =Operation Mode Select Program
AUTHOR : HMC
FAMILY : Mode
NAME : Mode
VERSION : 1.0


VAR_INPUT
  SSD_Manual : BOOL ;
  SSD_Auto : BOOL ;
  PB_Ready : BOOL ;
  PB_Auto_Run : BOOL ;
  PB_Remote_Ready : BOOL ;
  PB_Remote_Auto_Run : BOOL ;
  PB_Lamp_CHK : BOOL ;
  M_Air_Error : BOOL ;
  M_Water_Error : BOOL ;
  M_Total_Error : BOOL ;
  M_EStop : BOOL ;
  EXT_Ready : BOOL ;
  EXT_Auto : BOOL ;
  T_SemiAuto : TIME ;
  M_FLICK : BOOL ;
END_VAR
VAR_OUTPUT
  M_Ready_On : BOOL ;
  M_Auto_Mode : BOOL ;
  M_SemiAuto_Mode : BOOL ;
  M_Manual_Mode : BOOL ;
  M_Auto_Run : BOOL ;
  LP_Ready_On : BOOL ;
  LP_Auto_Run : BOOL ;
END_VAR
VAR
  AUTO_MODE_DELAY : SFB 4;
  SEMI_AUTO_DELAY : SFB 4;
  MANUAL_DELAY : SFB 4;
END_VAR
BEGIN
NETWORK
TITLE =Auto Mode Select Program
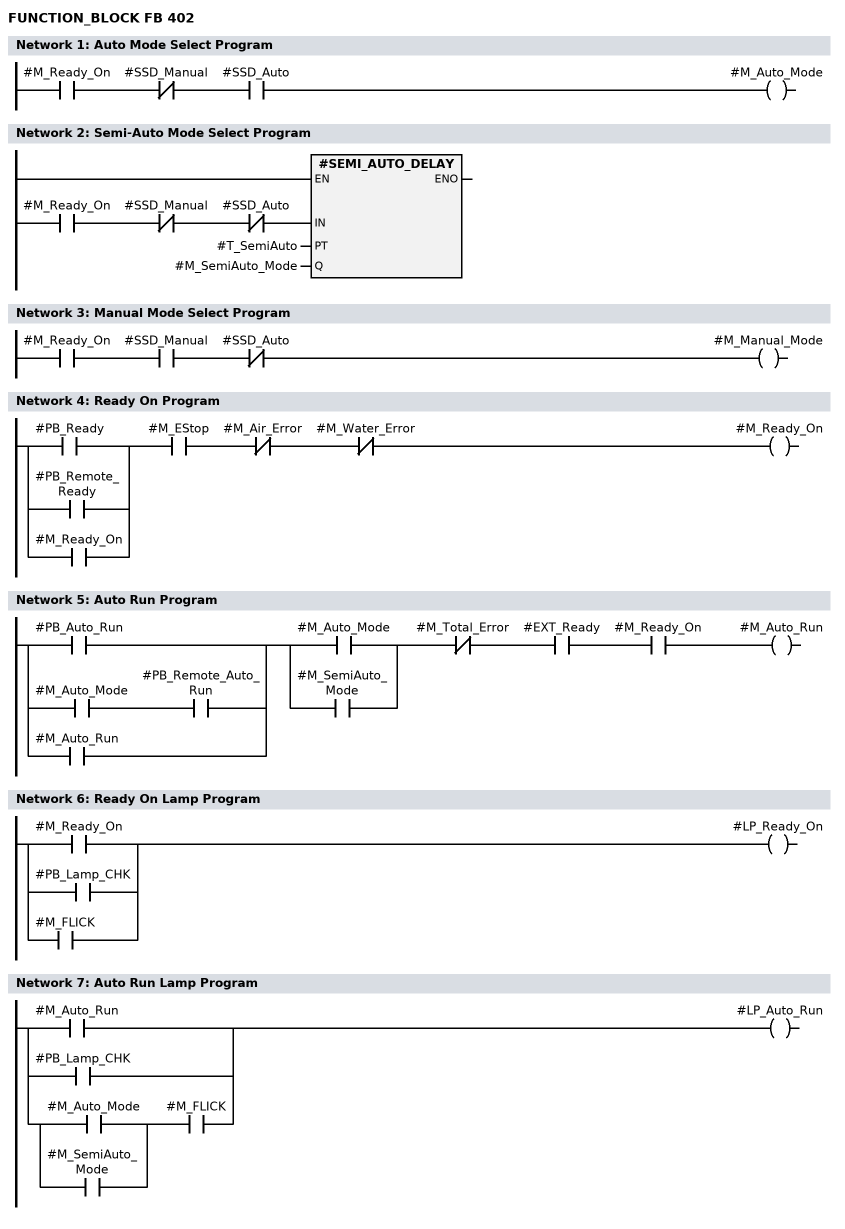

      A     #M_Ready_On;
      AN    #SSD_Manual;
      A     #SSD_Auto;
      =     #M_Auto_Mode;
NETWORK
TITLE =Semi-Auto Mode Select Program

      A     #M_Ready_On;
      AN    #SSD_Manual;
      AN    #SSD_Auto;
      =     L      0.0;
      BLD   103;
      CALL #SEMI_AUTO_DELAY (
           IN                       := L      0.0,
           PT                       := #T_SemiAuto,
           Q                        := #M_SemiAuto_Mode);

      NOP   0;
NETWORK
TITLE =Manual Mode Select Program

      A     #M_Ready_On;
      A     #SSD_Manual;
      AN    #SSD_Auto;
      =     #M_Manual_Mode;
NETWORK
TITLE =Ready On Program

      A(    ;
      O     #PB_Ready;
      O     #PB_Remote_Ready;
      O     #M_Ready_On;
      )     ;
      A     #M_EStop;
      AN    #M_Air_Error;
      AN    #M_Water_Error;
      =     #M_Ready_On;
NETWORK
TITLE =Auto Run Program

      A(    ;
      O     #PB_Auto_Run;
      O     ;
      A     #M_Auto_Mode;
      A     #PB_Remote_Auto_Run;
      O     #M_Auto_Run;
      )     ;
      A(    ;
      O     #M_Auto_Mode;
      O     #M_SemiAuto_Mode;
      )     ;
      AN    #M_Total_Error;
      A     #EXT_Ready;
      A     #M_Ready_On;
      =     #M_Auto_Run;
NETWORK
TITLE =Ready On Lamp Program

      O     #M_Ready_On;
      O     #PB_Lamp_CHK;
      O     #M_FLICK;
      =     #LP_Ready_On;
NETWORK
TITLE =Auto Run Lamp Program

      O     #M_Auto_Run;
      O     #PB_Lamp_CHK;
      O     ;
      A(    ;
      O     #M_Auto_Mode;
      O     #M_SemiAuto_Mode;
      )     ;
      A     #M_FLICK;
      =     #LP_Auto_Run;
END_FUNCTION_BLOCK

FUNCTION_BLOCK FB 424
TITLE =Sensor Error,Lamp Variables Program
AUTHOR : HMC
FAMILY : Common
NAME : Common
VERSION : 1.0


VAR_INPUT
  Enable_Aux : BOOL ;
  Adv_Amount : INT ;
  Ret_Amount : INT ;
  LS_Adv1 : BOOL ;
  LS_Ret1 : BOOL ;
  LS_Adv2 : BOOL ;
  LS_Ret2 : BOOL ;
  LS_Adv3 : BOOL ;
  LS_Ret3 : BOOL ;
  LS_Adv4 : BOOL ;
  LS_Ret4 : BOOL ;
  SOL_Adv : BOOL ;
  SOL_Ret : BOOL ;
  M_Ready : BOOL ;
  T_CHK1 : TIME ;
  T_CHK2 : TIME ;
  PB_Lamp_CHK : BOOL ;
  PB_Error_Rst : BOOL ;
  M_FLICK : BOOL ;
END_VAR
VAR_OUTPUT
  M_Adv_Err : BOOL ;
  M_Ret_Err : BOOL ;
  LP_Adv : BOOL ;
  LP_Ret : BOOL ;
  Visu_Adv : WORD ;
  Visu_Ret : WORD ;
END_VAR
VAR
  Error_T1 : SFB 4;
  Error_T2 : SFB 4;
  CHK_Aux1 : BOOL ;
  CHK_Aux2 : BOOL ;
  Error_T1_DN : BOOL ;
  Error_T2_DN : BOOL ;
  Adv_Memo : BOOL ;
  Visu_Adv_Arr : ARRAY  [0 .. 15 ] OF BOOL ;
  Visu_Ret_Arr : ARRAY  [0 .. 15 ] OF BOOL ;
  BLK_Move_Ret : INT ;
  Enable : BOOL ;
  Adv_End : BOOL ;
  Ret_End : BOOL ;
END_VAR
BEGIN
NETWORK
TITLE =
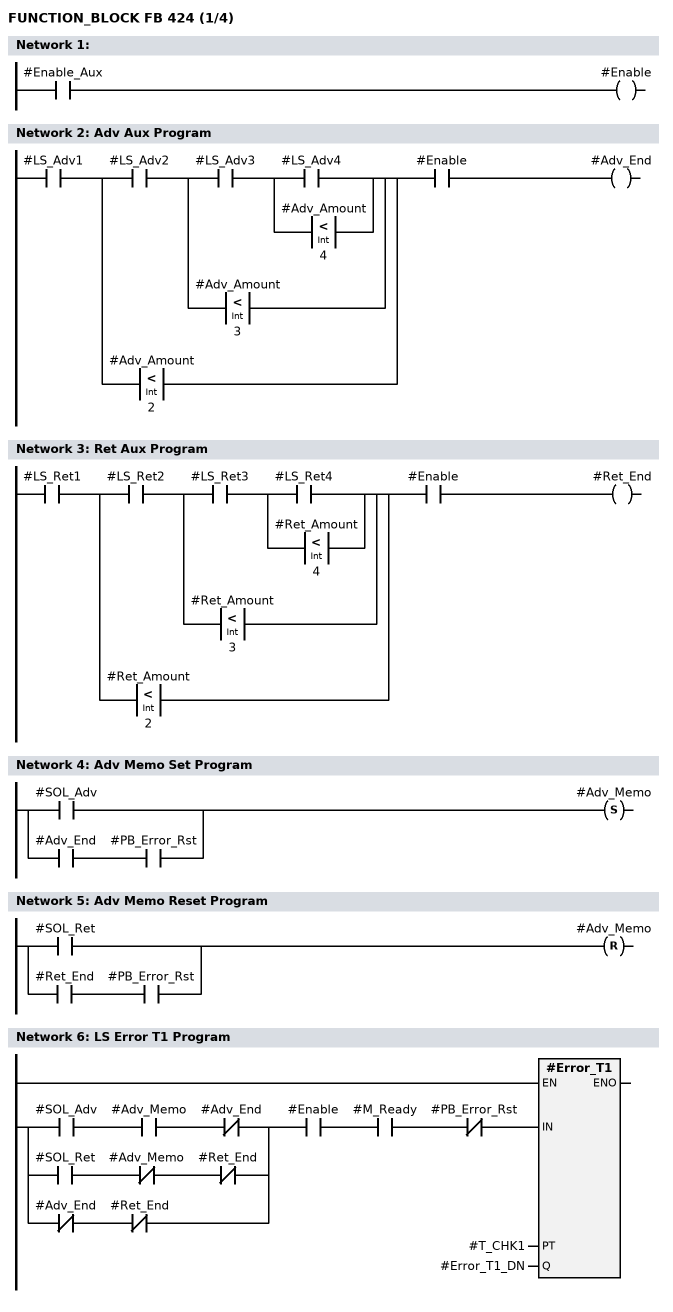

      A     #Enable_Aux;
      =     #Enable;
NETWORK
TITLE =Adv Aux Program

      A     #LS_Adv1;
      A(    ;
      A     #LS_Adv2;
      A(    ;
      A     #LS_Adv3;
      A(    ;
      O     #LS_Adv4;
      O(    ;
      L     #Adv_Amount;
      L     4;
      <I    ;
      )     ;
      )     ;
      O(    ;
      L     #Adv_Amount;
      L     3;
      <I    ;
      )     ;
      )     ;
      O(    ;
      L     #Adv_Amount;
      L     2;
      <I    ;
      )     ;
      )     ;
      A     #Enable;
      =     #Adv_End;
NETWORK
TITLE =Ret Aux Program

      A     #LS_Ret1;
      A(    ;
      A     #LS_Ret2;
      A(    ;
      A     #LS_Ret3;
      A(    ;
      O     #LS_Ret4;
      O(    ;
      L     #Ret_Amount;
      L     4;
      <I    ;
      )     ;
      )     ;
      O(    ;
      L     #Ret_Amount;
      L     3;
      <I    ;
      )     ;
      )     ;
      O(    ;
      L     #Ret_Amount;
      L     2;
      <I    ;
      )     ;
      )     ;
      A     #Enable;
      =     #Ret_End;
NETWORK
TITLE =Adv Memo Set Program

      O     #SOL_Adv;
      O     ;
      A     #Adv_End;
      A     #PB_Error_Rst;
      S     #Adv_Memo;
NETWORK
TITLE =Adv Memo Reset Program

      O     #SOL_Ret;
      O     ;
      A     #Ret_End;
      A     #PB_Error_Rst;
      R     #Adv_Memo;
NETWORK
TITLE =LS Error T1 Program

      A(    ;
      A     #SOL_Adv;
      A     #Adv_Memo;
      AN    #Adv_End;
      O     ;
      A     #SOL_Ret;
      AN    #Adv_Memo;
      AN    #Ret_End;
      O     ;
      AN    #Adv_End;
      AN    #Ret_End;
      )     ;
      A     #Enable;
      A     #M_Ready;
      AN    #PB_Error_Rst;
      =     L      0.0;
      BLD   103;
      CALL #Error_T1 (
           IN                       := L      0.0,
           PT                       := #T_CHK1,
           Q                        := #Error_T1_DN);

      NOP   0;
NETWORK
TITLE =Check Aux1 Program
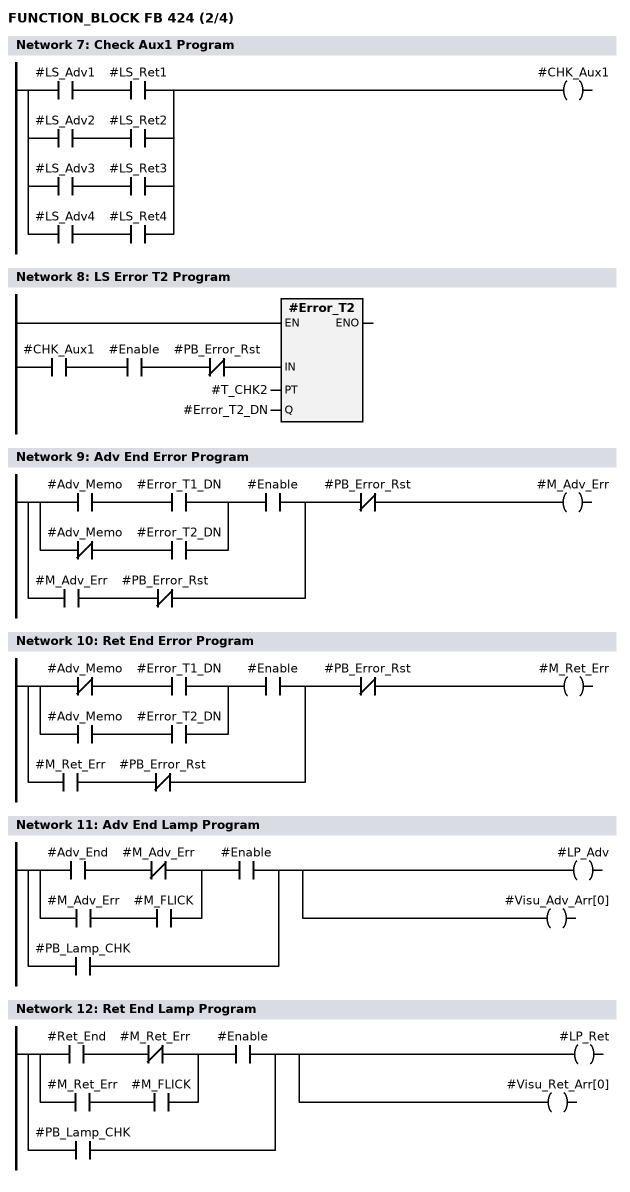

      A     #LS_Adv1;
      A     #LS_Ret1;
      O     ;
      A     #LS_Adv2;
      A     #LS_Ret2;
      O     ;
      A     #LS_Adv3;
      A     #LS_Ret3;
      O     ;
      A     #LS_Adv4;
      A     #LS_Ret4;
      =     #CHK_Aux1;
NETWORK
TITLE =LS Error T2 Program

      A     #CHK_Aux1;
      A     #Enable;
      AN    #PB_Error_Rst;
      =     L      0.0;
      BLD   103;
      CALL #Error_T2 (
           IN                       := L      0.0,
           PT                       := #T_CHK2,
           Q                        := #Error_T2_DN);

      NOP   0;
NETWORK
TITLE =Adv End Error Program

      A(    ;
      A(    ;
      A     #Adv_Memo;
      A     #Error_T1_DN;
      O     ;
      AN    #Adv_Memo;
      A     #Error_T2_DN;
      )     ;
      A     #Enable;
      O     ;
      A     #M_Adv_Err;
      AN    #PB_Error_Rst;
      )     ;
      AN    #PB_Error_Rst;
      =     #M_Adv_Err;
NETWORK
TITLE =Ret End Error Program

      A(    ;
      A(    ;
      AN    #Adv_Memo;
      A     #Error_T1_DN;
      O     ;
      A     #Adv_Memo;
      A     #Error_T2_DN;
      )     ;
      A     #Enable;
      O     ;
      A     #M_Ret_Err;
      AN    #PB_Error_Rst;
      )     ;
      AN    #PB_Error_Rst;
      =     #M_Ret_Err;
NETWORK
TITLE =Adv End Lamp Program

      A(    ;
      A     #Adv_End;
      AN    #M_Adv_Err;
      O     ;
      A     #M_Adv_Err;
      A     #M_FLICK;
      )     ;
      A     #Enable;
      O     #PB_Lamp_CHK;
      =     #LP_Adv;
      =     #Visu_Adv_Arr[0];
NETWORK
TITLE =Ret End Lamp Program

      A(    ;
      A     #Ret_End;
      AN    #M_Ret_Err;
      O     ;
      A     #M_Ret_Err;
      A     #M_FLICK;
      )     ;
      A     #Enable;
      O     #PB_Lamp_CHK;
      =     #LP_Ret;
      =     #Visu_Ret_Arr[0];
NETWORK
TITLE =Adv LS_1 Lamp Program
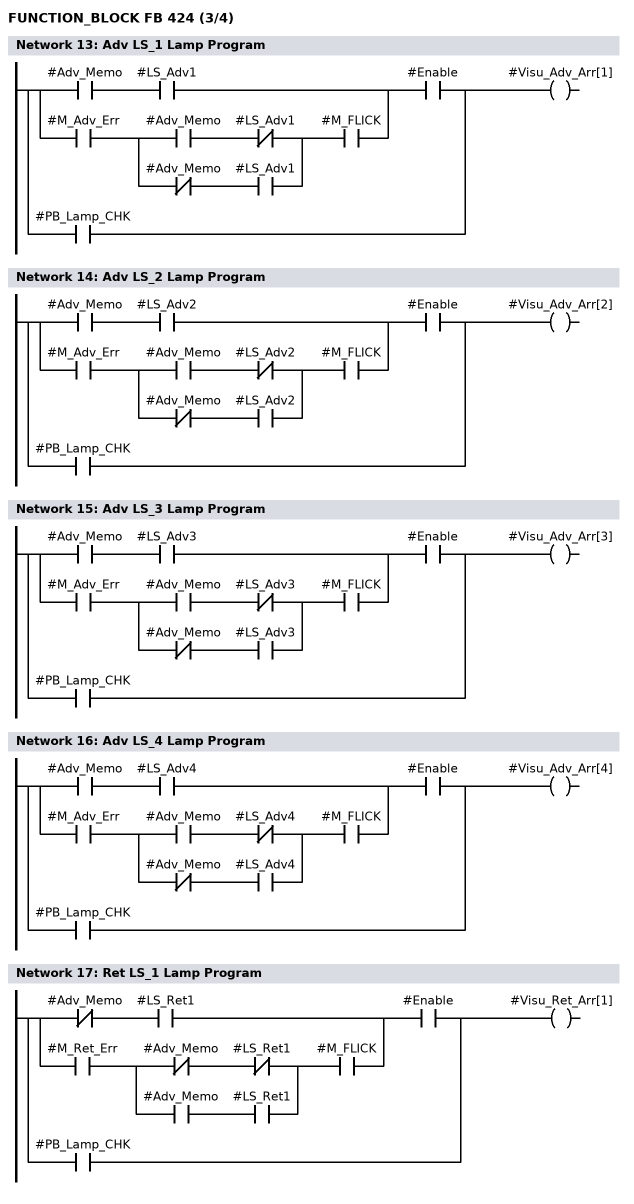

      A(    ;
      A     #Adv_Memo;
      A     #LS_Adv1;
      O     ;
      A     #M_Adv_Err;
      A(    ;
      A     #Adv_Memo;
      AN    #LS_Adv1;
      O     ;
      AN    #Adv_Memo;
      A     #LS_Adv1;
      )     ;
      A     #M_FLICK;
      )     ;
      A     #Enable;
      O     #PB_Lamp_CHK;
      =     #Visu_Adv_Arr[1];
NETWORK
TITLE =Adv LS_2 Lamp Program
//
//
      A(    ;
      A     #Adv_Memo;
      A     #LS_Adv2;
      O     ;
      A     #M_Adv_Err;
      A(    ;
      A     #Adv_Memo;
      AN    #LS_Adv2;
      O     ;
      AN    #Adv_Memo;
      A     #LS_Adv2;
      )     ;
      A     #M_FLICK;
      )     ;
      A     #Enable;
      O     #PB_Lamp_CHK;
      =     #Visu_Adv_Arr[2];
NETWORK
TITLE =Adv LS_3 Lamp Program
//
//
      A(    ;
      A     #Adv_Memo;
      A     #LS_Adv3;
      O     ;
      A     #M_Adv_Err;
      A(    ;
      A     #Adv_Memo;
      AN    #LS_Adv3;
      O     ;
      AN    #Adv_Memo;
      A     #LS_Adv3;
      )     ;
      A     #M_FLICK;
      )     ;
      A     #Enable;
      O     #PB_Lamp_CHK;
      =     #Visu_Adv_Arr[3];
NETWORK
TITLE =Adv LS_4 Lamp Program
//
//
      A(    ;
      A     #Adv_Memo;
      A     #LS_Adv4;
      O     ;
      A     #M_Adv_Err;
      A(    ;
      A     #Adv_Memo;
      AN    #LS_Adv4;
      O     ;
      AN    #Adv_Memo;
      A     #LS_Adv4;
      )     ;
      A     #M_FLICK;
      )     ;
      A     #Enable;
      O     #PB_Lamp_CHK;
      =     #Visu_Adv_Arr[4];
NETWORK
TITLE =Ret LS_1 Lamp Program
//
//
      A(    ;
      AN    #Adv_Memo;
      A     #LS_Ret1;
      O     ;
      A     #M_Ret_Err;
      A(    ;
      AN    #Adv_Memo;
      AN    #LS_Ret1;
      O     ;
      A     #Adv_Memo;
      A     #LS_Ret1;
      )     ;
      A     #M_FLICK;
      )     ;
      A     #Enable;
      O     #PB_Lamp_CHK;
      =     #Visu_Ret_Arr[1];
NETWORK
TITLE =Ret LS_2 Lamp Program
//
//
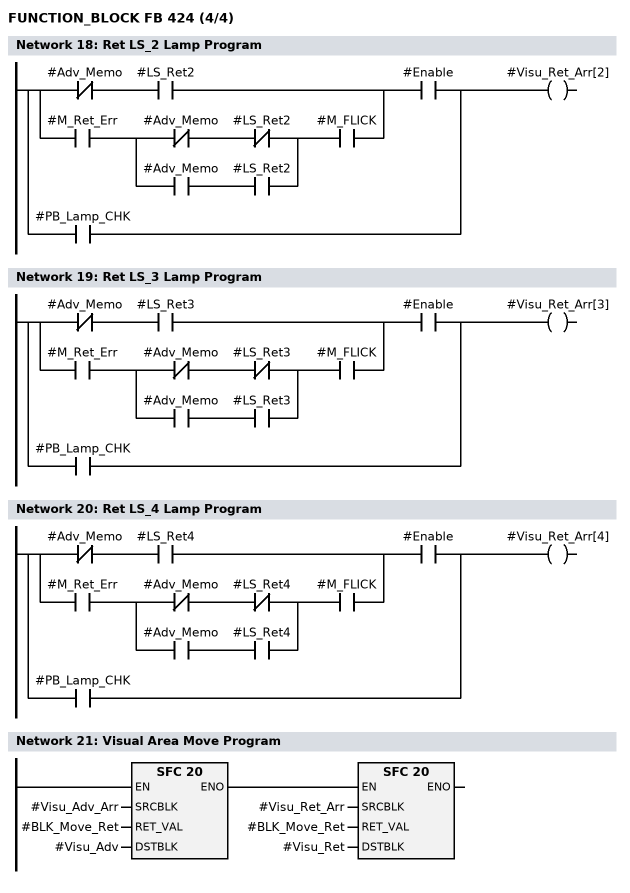
      A(    ;
      AN    #Adv_Memo;
      A     #LS_Ret2;
      O     ;
      A     #M_Ret_Err;
      A(    ;
      AN    #Adv_Memo;
      AN    #LS_Ret2;
      O     ;
      A     #Adv_Memo;
      A     #LS_Ret2;
      )     ;
      A     #M_FLICK;
      )     ;
      A     #Enable;
      O     #PB_Lamp_CHK;
      =     #Visu_Ret_Arr[2];
NETWORK
TITLE =Ret LS_3 Lamp Program
//
//
      A(    ;
      AN    #Adv_Memo;
      A     #LS_Ret3;
      O     ;
      A     #M_Ret_Err;
      A(    ;
      AN    #Adv_Memo;
      AN    #LS_Ret3;
      O     ;
      A     #Adv_Memo;
      A     #LS_Ret3;
      )     ;
      A     #M_FLICK;
      )     ;
      A     #Enable;
      O     #PB_Lamp_CHK;
      =     #Visu_Ret_Arr[3];
NETWORK
TITLE =Ret LS_4 Lamp Program
//
//
      A(    ;
      AN    #Adv_Memo;
      A     #LS_Ret4;
      O     ;
      A     #M_Ret_Err;
      A(    ;
      AN    #Adv_Memo;
      AN    #LS_Ret4;
      O     ;
      A     #Adv_Memo;
      A     #LS_Ret4;
      )     ;
      A     #M_FLICK;
      )     ;
      A     #Enable;
      O     #PB_Lamp_CHK;
      =     #Visu_Ret_Arr[4];
NETWORK
TITLE =Visual Area Move Program

      A(    ;
      CALL SFC   20 (
           SRCBLK                   := #Visu_Adv_Arr,
           RET_VAL                  := #BLK_Move_Ret,
           DSTBLK                   := #Visu_Adv);
      A     BR;
      )     ;
      JNB   _001;
      CALL SFC   20 (
           SRCBLK                   := #Visu_Ret_Arr,
           RET_VAL                  := #BLK_Move_Ret,
           DSTBLK                   := #Visu_Ret);
_001: NOP   0;
END_FUNCTION_BLOCK

FUNCTION_BLOCK FB 430
TITLE =Sensor End,Error,Lamp Variables Program
AUTHOR : HMC
FAMILY : Common
NAME : Common
VERSION : 1.0


VAR_INPUT
  General_JIG : BOOL ;
  DAECHA_ID_ON : BOOL ;
  M_Ready : BOOL ;
  SOL_Adv : BOOL ;
  SOL_Ret : BOOL ;
  Adv_Amount : INT ;
  Ret_Amount : INT ;
  LS_Adv1 : BOOL ;
  LS_Ret1 : BOOL ;
  LS_Adv2 : BOOL ;
  LS_Ret2 : BOOL ;
  LS_Adv3 : BOOL ;
  LS_Ret3 : BOOL ;
  LS_Adv4 : BOOL ;
  LS_Ret4 : BOOL ;
  LS_Adv5 : BOOL ;
  LS_Ret5 : BOOL ;
  LS_Adv6 : BOOL ;
  LS_Ret6 : BOOL ;
  LS_Adv7 : BOOL ;
  LS_Ret7 : BOOL ;
  LS_Adv8 : BOOL ;
  LS_Ret8 : BOOL ;
  LS_Adv9 : BOOL ;
  LS_Ret9 : BOOL ;
  LS_Adv10 : BOOL ;
  LS_Ret10 : BOOL ;
  T_CHK1 : TIME ;
  T_CHK2 : TIME ;
  PB_Error_Rst : BOOL ;
  PB_Lamp_CHK : BOOL ;
  M_FLICK : BOOL ;
END_VAR
VAR_OUTPUT
  M_Adv_Err : BOOL ;
  M_Ret_Err : BOOL ;
  LP_Adv : BOOL ;
  LP_Ret : BOOL ;
  Visu_Adv : WORD ;
  Visu_Ret : WORD ;
END_VAR
VAR
  Error_T1 : SFB 4;
  Error_T2 : SFB 4;
  Adv_End_Delay : SFB 4;
  Ret_End_Delay : SFB 4;
  Adv_End_Aux : BOOL ;
  Ret_End_Aux : BOOL ;
  CHK_Aux1 : BOOL ;
  CHK_Aux2 : BOOL ;
  Error_T1_DN : BOOL ;
  Error_T2_DN : BOOL ;
  Adv_Memo : BOOL ;
  Visu_Adv_Arr : ARRAY  [0 .. 15 ] OF BOOL ;
  Visu_Ret_Arr : ARRAY  [0 .. 15 ] OF BOOL ;
  BLK_Move_Ret : INT ;
  Enable : BOOL ;
  M_Adv_End : BOOL ;
  M_Ret_End : BOOL ;
END_VAR
BEGIN
NETWORK
TITLE =
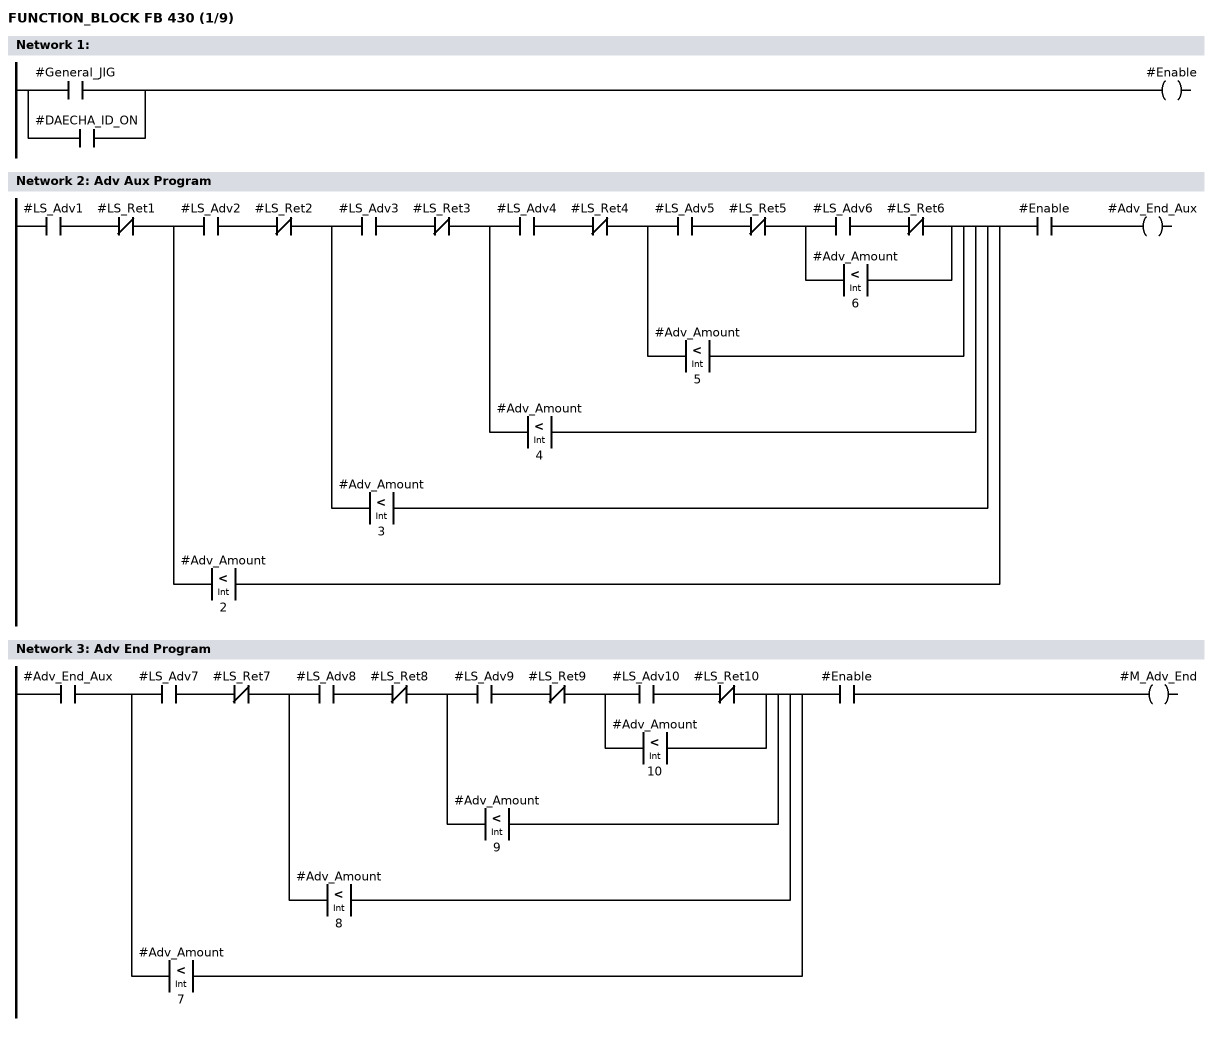

      O     #General_JIG;
      O     #DAECHA_ID_ON;
      =     #Enable;
NETWORK
TITLE =Adv Aux Program

      A     #LS_Adv1;
      AN    #LS_Ret1;
      A(    ;
      A     #LS_Adv2;
      AN    #LS_Ret2;
      A(    ;
      A     #LS_Adv3;
      AN    #LS_Ret3;
      A(    ;
      A     #LS_Adv4;
      AN    #LS_Ret4;
      A(    ;
      A     #LS_Adv5;
      AN    #LS_Ret5;
      A(    ;
      A     #LS_Adv6;
      AN    #LS_Ret6;
      O(    ;
      L     #Adv_Amount;
      L     6;
      <I    ;
      )     ;
      )     ;
      O(    ;
      L     #Adv_Amount;
      L     5;
      <I    ;
      )     ;
      )     ;
      O(    ;
      L     #Adv_Amount;
      L     4;
      <I    ;
      )     ;
      )     ;
      O(    ;
      L     #Adv_Amount;
      L     3;
      <I    ;
      )     ;
      )     ;
      O(    ;
      L     #Adv_Amount;
      L     2;
      <I    ;
      )     ;
      )     ;
      A     #Enable;
      =     #Adv_End_Aux;
NETWORK
TITLE =Adv End Program

      A     #Adv_End_Aux;
      A(    ;
      A     #LS_Adv7;
      AN    #LS_Ret7;
      A(    ;
      A     #LS_Adv8;
      AN    #LS_Ret8;
      A(    ;
      A     #LS_Adv9;
      AN    #LS_Ret9;
      A(    ;
      A     #LS_Adv10;
      AN    #LS_Ret10;
      O(    ;
      L     #Adv_Amount;
      L     10;
      <I    ;
      )     ;
      )     ;
      O(    ;
      L     #Adv_Amount;
      L     9;
      <I    ;
      )     ;
      )     ;
      O(    ;
      L     #Adv_Amount;
      L     8;
      <I    ;
      )     ;
      )     ;
      O(    ;
      L     #Adv_Amount;
      L     7;
      <I    ;
      )     ;
      )     ;
      A     #Enable;
      =     #M_Adv_End;
NETWORK
TITLE =Ret Aux Program
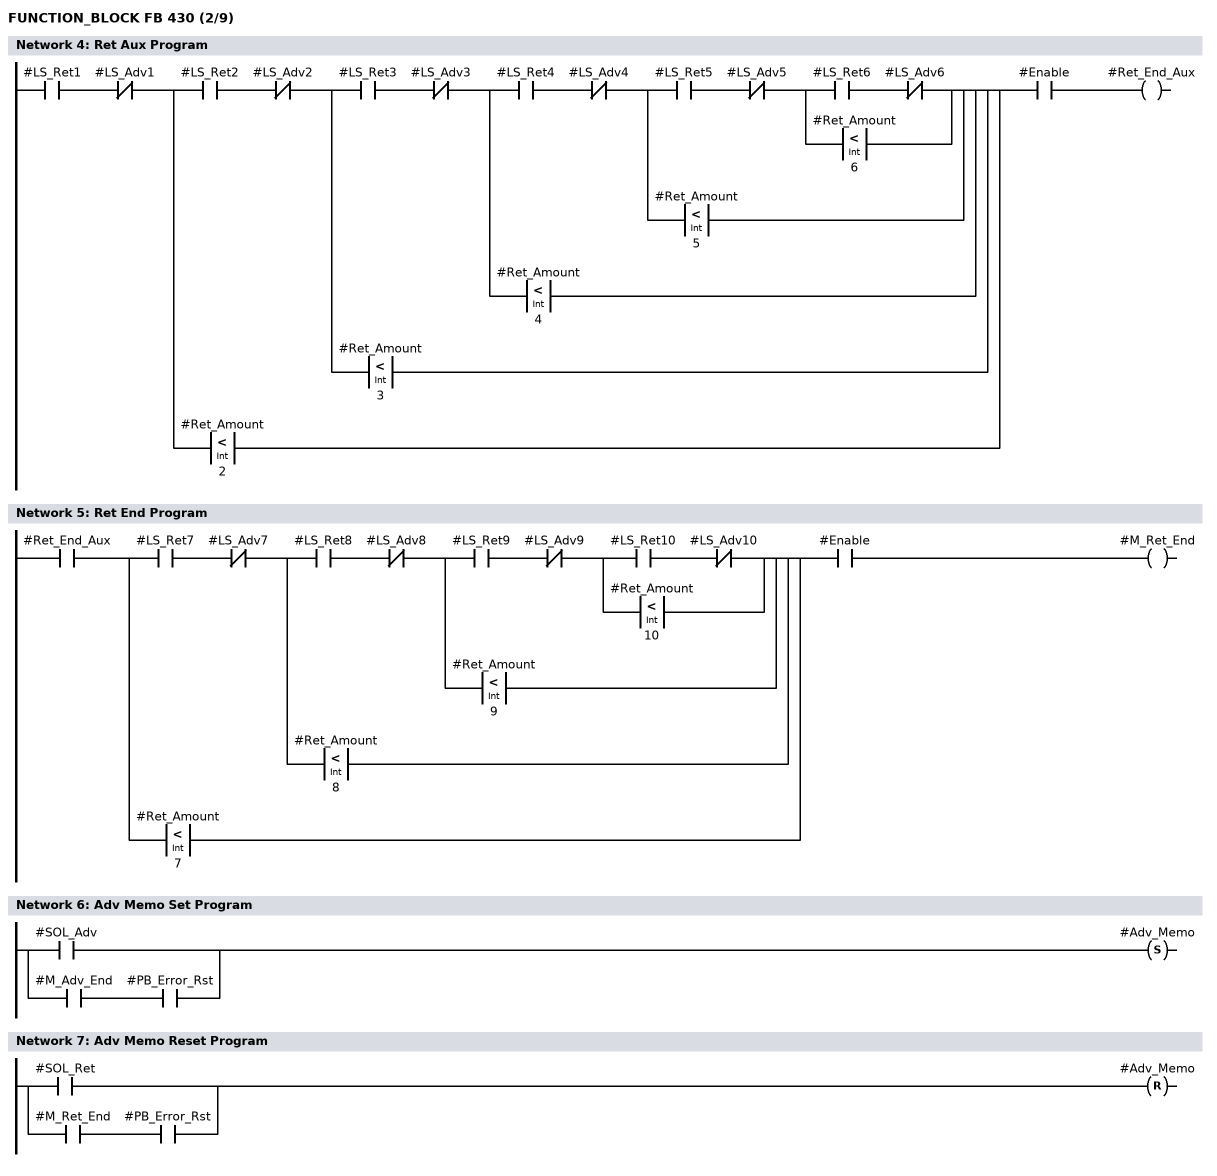

      A     #LS_Ret1;
      AN    #LS_Adv1;
      A(    ;
      A     #LS_Ret2;
      AN    #LS_Adv2;
      A(    ;
      A     #LS_Ret3;
      AN    #LS_Adv3;
      A(    ;
      A     #LS_Ret4;
      AN    #LS_Adv4;
      A(    ;
      A     #LS_Ret5;
      AN    #LS_Adv5;
      A(    ;
      A     #LS_Ret6;
      AN    #LS_Adv6;
      O(    ;
      L     #Ret_Amount;
      L     6;
      <I    ;
      )     ;
      )     ;
      O(    ;
      L     #Ret_Amount;
      L     5;
      <I    ;
      )     ;
      )     ;
      O(    ;
      L     #Ret_Amount;
      L     4;
      <I    ;
      )     ;
      )     ;
      O(    ;
      L     #Ret_Amount;
      L     3;
      <I    ;
      )     ;
      )     ;
      O(    ;
      L     #Ret_Amount;
      L     2;
      <I    ;
      )     ;
      )     ;
      A     #Enable;
      =     #Ret_End_Aux;
NETWORK
TITLE =Ret End Program

      A     #Ret_End_Aux;
      A(    ;
      A     #LS_Ret7;
      AN    #LS_Adv7;
      A(    ;
      A     #LS_Ret8;
      AN    #LS_Adv8;
      A(    ;
      A     #LS_Ret9;
      AN    #LS_Adv9;
      A(    ;
      A     #LS_Ret10;
      AN    #LS_Adv10;
      O(    ;
      L     #Ret_Amount;
      L     10;
      <I    ;
      )     ;
      )     ;
      O(    ;
      L     #Ret_Amount;
      L     9;
      <I    ;
      )     ;
      )     ;
      O(    ;
      L     #Ret_Amount;
      L     8;
      <I    ;
      )     ;
      )     ;
      O(    ;
      L     #Ret_Amount;
      L     7;
      <I    ;
      )     ;
      )     ;
      A     #Enable;
      =     #M_Ret_End;
NETWORK
TITLE =Adv Memo Set Program

      O     #SOL_Adv;
      O     ;
      A     #M_Adv_End;
      A     #PB_Error_Rst;
      S     #Adv_Memo;
NETWORK
TITLE =Adv Memo Reset Program

      O     #SOL_Ret;
      O     ;
      A     #M_Ret_End;
      A     #PB_Error_Rst;
      R     #Adv_Memo;
NETWORK
TITLE =LS Error T1 Program
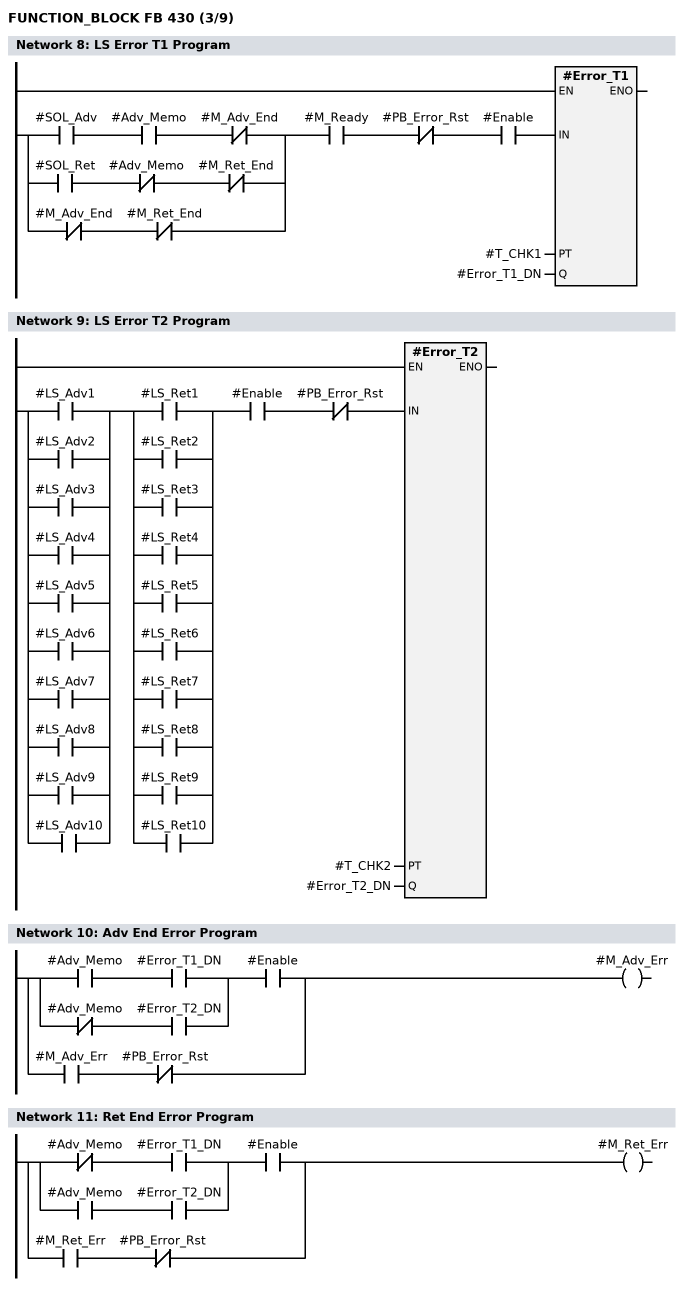

      A(    ;
      A     #SOL_Adv;
      A     #Adv_Memo;
      AN    #M_Adv_End;
      O     ;
      A     #SOL_Ret;
      AN    #Adv_Memo;
      AN    #M_Ret_End;
      O     ;
      AN    #M_Adv_End;
      AN    #M_Ret_End;
      )     ;
      A     #M_Ready;
      AN    #PB_Error_Rst;
      A     #Enable;
      =     L      0.0;
      BLD   103;
      CALL #Error_T1 (
           IN                       := L      0.0,
           PT                       := #T_CHK1,
           Q                        := #Error_T1_DN);

      NOP   0;
NETWORK
TITLE =LS Error T2 Program

      A(    ;
      O     #LS_Adv1;
      O     #LS_Adv2;
      O     #LS_Adv3;
      O     #LS_Adv4;
      O     #LS_Adv5;
      O     #LS_Adv6;
      O     #LS_Adv7;
      O     #LS_Adv8;
      O     #LS_Adv9;
      O     #LS_Adv10;
      )     ;
      A(    ;
      O     #LS_Ret1;
      O     #LS_Ret2;
      O     #LS_Ret3;
      O     #LS_Ret4;
      O     #LS_Ret5;
      O     #LS_Ret6;
      O     #LS_Ret7;
      O     #LS_Ret8;
      O     #LS_Ret9;
      O     #LS_Ret10;
      )     ;
      A     #Enable;
      AN    #PB_Error_Rst;
      =     L      0.0;
      BLD   103;
      CALL #Error_T2 (
           IN                       := L      0.0,
           PT                       := #T_CHK2,
           Q                        := #Error_T2_DN);

      NOP   0;
NETWORK
TITLE =Adv End Error Program

      A(    ;
      A     #Adv_Memo;
      A     #Error_T1_DN;
      O     ;
      AN    #Adv_Memo;
      A     #Error_T2_DN;
      )     ;
      A     #Enable;
      O     ;
      A     #M_Adv_Err;
      AN    #PB_Error_Rst;
      =     #M_Adv_Err;
NETWORK
TITLE =Ret End Error Program

      A(    ;
      AN    #Adv_Memo;
      A     #Error_T1_DN;
      O     ;
      A     #Adv_Memo;
      A     #Error_T2_DN;
      )     ;
      A     #Enable;
      O     ;
      A     #M_Ret_Err;
      AN    #PB_Error_Rst;
      =     #M_Ret_Err;
NETWORK
TITLE =Adv End Lamp Program
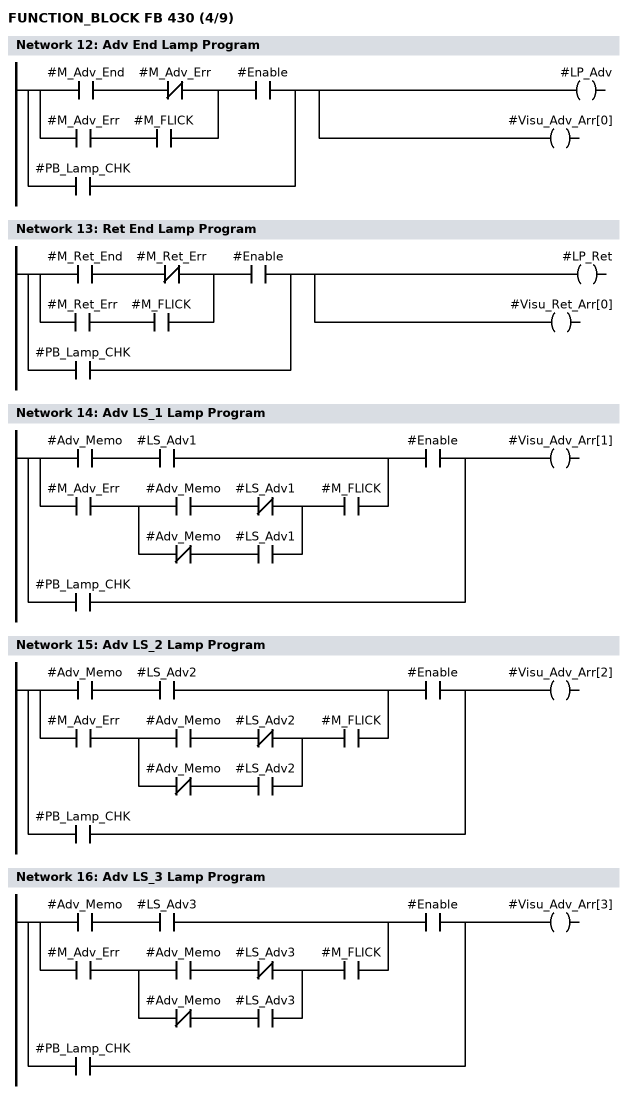

      A(    ;
      A     #M_Adv_End;
      AN    #M_Adv_Err;
      O     ;
      A     #M_Adv_Err;
      A     #M_FLICK;
      )     ;
      A     #Enable;
      O     #PB_Lamp_CHK;
      =     #LP_Adv;
      =     #Visu_Adv_Arr[0];
NETWORK
TITLE =Ret End Lamp Program

      A(    ;
      A     #M_Ret_End;
      AN    #M_Ret_Err;
      O     ;
      A     #M_Ret_Err;
      A     #M_FLICK;
      )     ;
      A     #Enable;
      O     #PB_Lamp_CHK;
      =     #LP_Ret;
      =     #Visu_Ret_Arr[0];
NETWORK
TITLE =Adv LS_1 Lamp Program

      A(    ;
      A     #Adv_Memo;
      A     #LS_Adv1;
      O     ;
      A     #M_Adv_Err;
      A(    ;
      A     #Adv_Memo;
      AN    #LS_Adv1;
      O     ;
      AN    #Adv_Memo;
      A     #LS_Adv1;
      )     ;
      A     #M_FLICK;
      )     ;
      A     #Enable;
      O     #PB_Lamp_CHK;
      =     #Visu_Adv_Arr[1];
NETWORK
TITLE =Adv LS_2 Lamp Program
//
//
      A(    ;
      A     #Adv_Memo;
      A     #LS_Adv2;
      O     ;
      A     #M_Adv_Err;
      A(    ;
      A     #Adv_Memo;
      AN    #LS_Adv2;
      O     ;
      AN    #Adv_Memo;
      A     #LS_Adv2;
      )     ;
      A     #M_FLICK;
      )     ;
      A     #Enable;
      O     #PB_Lamp_CHK;
      =     #Visu_Adv_Arr[2];
NETWORK
TITLE =Adv LS_3 Lamp Program
//
//
      A(    ;
      A     #Adv_Memo;
      A     #LS_Adv3;
      O     ;
      A     #M_Adv_Err;
      A(    ;
      A     #Adv_Memo;
      AN    #LS_Adv3;
      O     ;
      AN    #Adv_Memo;
      A     #LS_Adv3;
      )     ;
      A     #M_FLICK;
      )     ;
      A     #Enable;
      O     #PB_Lamp_CHK;
      =     #Visu_Adv_Arr[3];
NETWORK
TITLE =Adv LS_4 Lamp Program
//
//
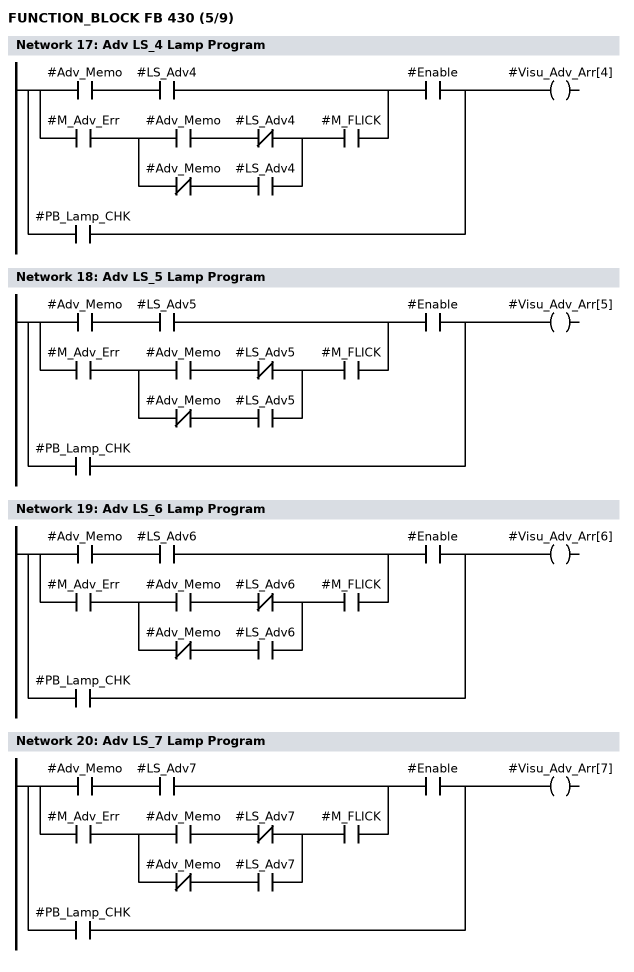
      A(    ;
      A     #Adv_Memo;
      A     #LS_Adv4;
      O     ;
      A     #M_Adv_Err;
      A(    ;
      A     #Adv_Memo;
      AN    #LS_Adv4;
      O     ;
      AN    #Adv_Memo;
      A     #LS_Adv4;
      )     ;
      A     #M_FLICK;
      )     ;
      A     #Enable;
      O     #PB_Lamp_CHK;
      =     #Visu_Adv_Arr[4];
NETWORK
TITLE =Adv LS_5 Lamp Program
//
//
      A(    ;
      A     #Adv_Memo;
      A     #LS_Adv5;
      O     ;
      A     #M_Adv_Err;
      A(    ;
      A     #Adv_Memo;
      AN    #LS_Adv5;
      O     ;
      AN    #Adv_Memo;
      A     #LS_Adv5;
      )     ;
      A     #M_FLICK;
      )     ;
      A     #Enable;
      O     #PB_Lamp_CHK;
      =     #Visu_Adv_Arr[5];
NETWORK
TITLE =Adv LS_6 Lamp Program
//
//
      A(    ;
      A     #Adv_Memo;
      A     #LS_Adv6;
      O     ;
      A     #M_Adv_Err;
      A(    ;
      A     #Adv_Memo;
      AN    #LS_Adv6;
      O     ;
      AN    #Adv_Memo;
      A     #LS_Adv6;
      )     ;
      A     #M_FLICK;
      )     ;
      A     #Enable;
      O     #PB_Lamp_CHK;
      =     #Visu_Adv_Arr[6];
NETWORK
TITLE =Adv LS_7 Lamp Program
//
//
      A(    ;
      A     #Adv_Memo;
      A     #LS_Adv7;
      O     ;
      A     #M_Adv_Err;
      A(    ;
      A     #Adv_Memo;
      AN    #LS_Adv7;
      O     ;
      AN    #Adv_Memo;
      A     #LS_Adv7;
      )     ;
      A     #M_FLICK;
      )     ;
      A     #Enable;
      O     #PB_Lamp_CHK;
      =     #Visu_Adv_Arr[7];
NETWORK
TITLE =Adv LS_8 Lamp Program
//
//
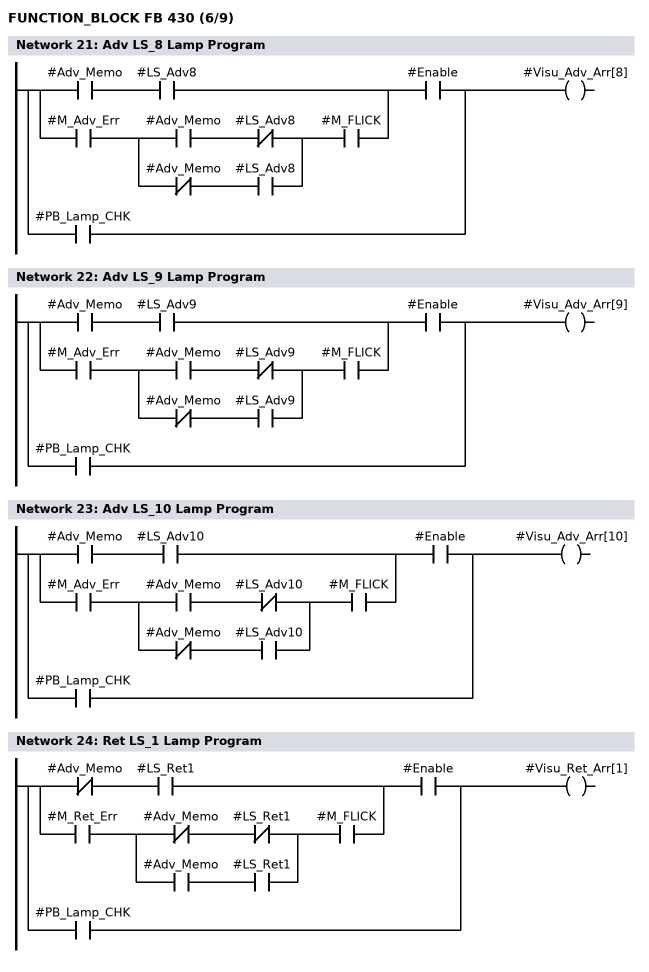
      A(    ;
      A     #Adv_Memo;
      A     #LS_Adv8;
      O     ;
      A     #M_Adv_Err;
      A(    ;
      A     #Adv_Memo;
      AN    #LS_Adv8;
      O     ;
      AN    #Adv_Memo;
      A     #LS_Adv8;
      )     ;
      A     #M_FLICK;
      )     ;
      A     #Enable;
      O     #PB_Lamp_CHK;
      =     #Visu_Adv_Arr[8];
NETWORK
TITLE =Adv LS_9 Lamp Program
//
//
      A(    ;
      A     #Adv_Memo;
      A     #LS_Adv9;
      O     ;
      A     #M_Adv_Err;
      A(    ;
      A     #Adv_Memo;
      AN    #LS_Adv9;
      O     ;
      AN    #Adv_Memo;
      A     #LS_Adv9;
      )     ;
      A     #M_FLICK;
      )     ;
      A     #Enable;
      O     #PB_Lamp_CHK;
      =     #Visu_Adv_Arr[9];
NETWORK
TITLE =Adv LS_10 Lamp Program
//
//
      A(    ;
      A     #Adv_Memo;
      A     #LS_Adv10;
      O     ;
      A     #M_Adv_Err;
      A(    ;
      A     #Adv_Memo;
      AN    #LS_Adv10;
      O     ;
      AN    #Adv_Memo;
      A     #LS_Adv10;
      )     ;
      A     #M_FLICK;
      )     ;
      A     #Enable;
      O     #PB_Lamp_CHK;
      =     #Visu_Adv_Arr[10];
NETWORK
TITLE =Ret LS_1 Lamp Program
//
//
      A(    ;
      AN    #Adv_Memo;
      A     #LS_Ret1;
      O     ;
      A     #M_Ret_Err;
      A(    ;
      AN    #Adv_Memo;
      AN    #LS_Ret1;
      O     ;
      A     #Adv_Memo;
      A     #LS_Ret1;
      )     ;
      A     #M_FLICK;
      )     ;
      A     #Enable;
      O     #PB_Lamp_CHK;
      =     #Visu_Ret_Arr[1];
NETWORK
TITLE =Ret LS_2 Lamp Program
//
//
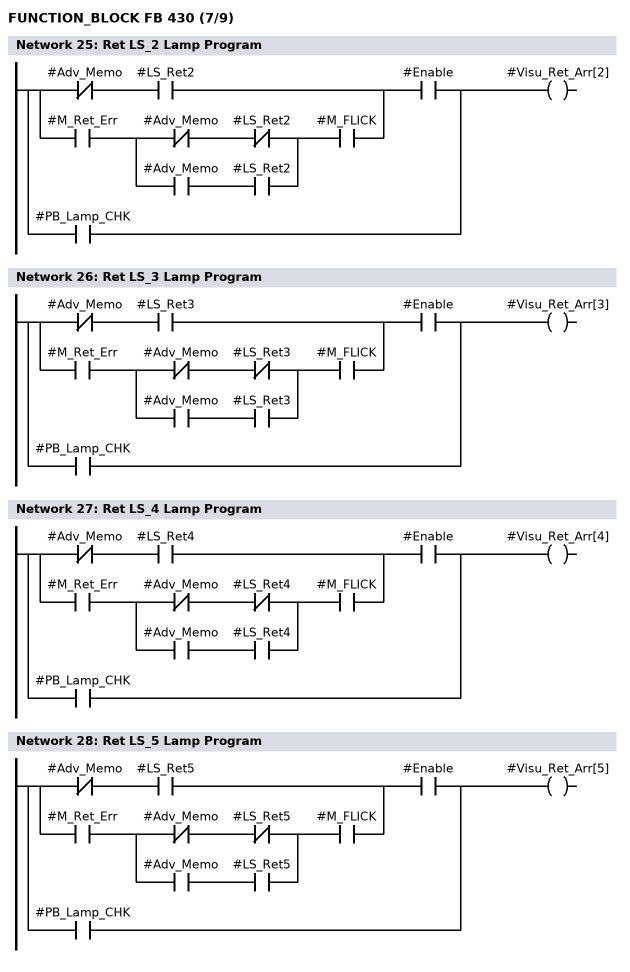
      A(    ;
      AN    #Adv_Memo;
      A     #LS_Ret2;
      O     ;
      A     #M_Ret_Err;
      A(    ;
      AN    #Adv_Memo;
      AN    #LS_Ret2;
      O     ;
      A     #Adv_Memo;
      A     #LS_Ret2;
      )     ;
      A     #M_FLICK;
      )     ;
      A     #Enable;
      O     #PB_Lamp_CHK;
      =     #Visu_Ret_Arr[2];
NETWORK
TITLE =Ret LS_3 Lamp Program
//
//
      A(    ;
      AN    #Adv_Memo;
      A     #LS_Ret3;
      O     ;
      A     #M_Ret_Err;
      A(    ;
      AN    #Adv_Memo;
      AN    #LS_Ret3;
      O     ;
      A     #Adv_Memo;
      A     #LS_Ret3;
      )     ;
      A     #M_FLICK;
      )     ;
      A     #Enable;
      O     #PB_Lamp_CHK;
      =     #Visu_Ret_Arr[3];
NETWORK
TITLE =Ret LS_4 Lamp Program
//
//
      A(    ;
      AN    #Adv_Memo;
      A     #LS_Ret4;
      O     ;
      A     #M_Ret_Err;
      A(    ;
      AN    #Adv_Memo;
      AN    #LS_Ret4;
      O     ;
      A     #Adv_Memo;
      A     #LS_Ret4;
      )     ;
      A     #M_FLICK;
      )     ;
      A     #Enable;
      O     #PB_Lamp_CHK;
      =     #Visu_Ret_Arr[4];
NETWORK
TITLE =Ret LS_5 Lamp Program
//
//
      A(    ;
      AN    #Adv_Memo;
      A     #LS_Ret5;
      O     ;
      A     #M_Ret_Err;
      A(    ;
      AN    #Adv_Memo;
      AN    #LS_Ret5;
      O     ;
      A     #Adv_Memo;
      A     #LS_Ret5;
      )     ;
      A     #M_FLICK;
      )     ;
      A     #Enable;
      O     #PB_Lamp_CHK;
      =     #Visu_Ret_Arr[5];
NETWORK
TITLE =Ret LS_6 Lamp Program
//
//
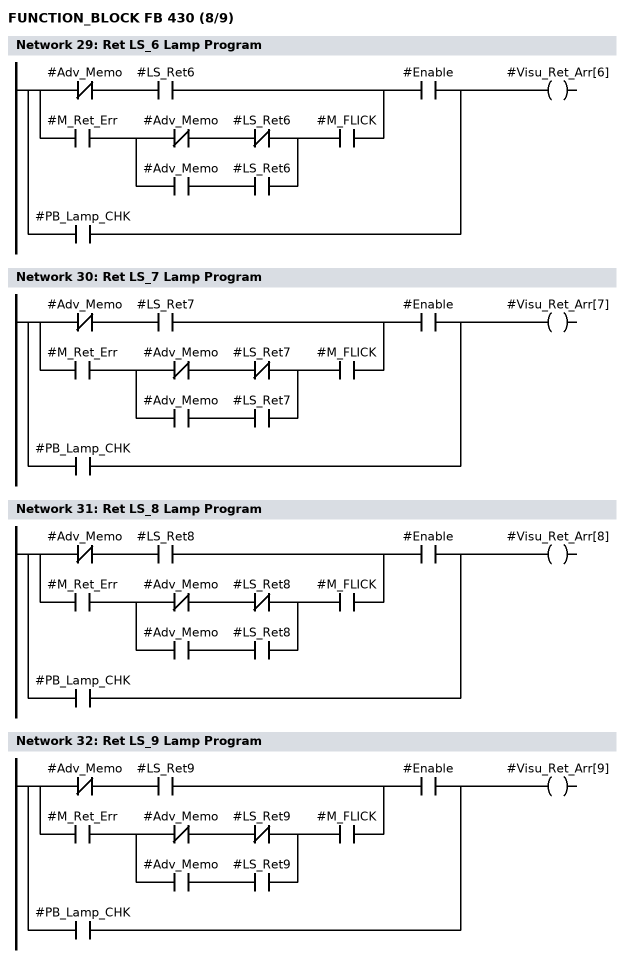
      A(    ;
      AN    #Adv_Memo;
      A     #LS_Ret6;
      O     ;
      A     #M_Ret_Err;
      A(    ;
      AN    #Adv_Memo;
      AN    #LS_Ret6;
      O     ;
      A     #Adv_Memo;
      A     #LS_Ret6;
      )     ;
      A     #M_FLICK;
      )     ;
      A     #Enable;
      O     #PB_Lamp_CHK;
      =     #Visu_Ret_Arr[6];
NETWORK
TITLE =Ret LS_7 Lamp Program
//
//
      A(    ;
      AN    #Adv_Memo;
      A     #LS_Ret7;
      O     ;
      A     #M_Ret_Err;
      A(    ;
      AN    #Adv_Memo;
      AN    #LS_Ret7;
      O     ;
      A     #Adv_Memo;
      A     #LS_Ret7;
      )     ;
      A     #M_FLICK;
      )     ;
      A     #Enable;
      O     #PB_Lamp_CHK;
      =     #Visu_Ret_Arr[7];
NETWORK
TITLE =Ret LS_8 Lamp Program
//
//
      A(    ;
      AN    #Adv_Memo;
      A     #LS_Ret8;
      O     ;
      A     #M_Ret_Err;
      A(    ;
      AN    #Adv_Memo;
      AN    #LS_Ret8;
      O     ;
      A     #Adv_Memo;
      A     #LS_Ret8;
      )     ;
      A     #M_FLICK;
      )     ;
      A     #Enable;
      O     #PB_Lamp_CHK;
      =     #Visu_Ret_Arr[8];
NETWORK
TITLE =Ret LS_9 Lamp Program
//
//
      A(    ;
      AN    #Adv_Memo;
      A     #LS_Ret9;
      O     ;
      A     #M_Ret_Err;
      A(    ;
      AN    #Adv_Memo;
      AN    #LS_Ret9;
      O     ;
      A     #Adv_Memo;
      A     #LS_Ret9;
      )     ;
      A     #M_FLICK;
      )     ;
      A     #Enable;
      O     #PB_Lamp_CHK;
      =     #Visu_Ret_Arr[9];
NETWORK
TITLE =Ret LS_10 Lamp Program
//
//
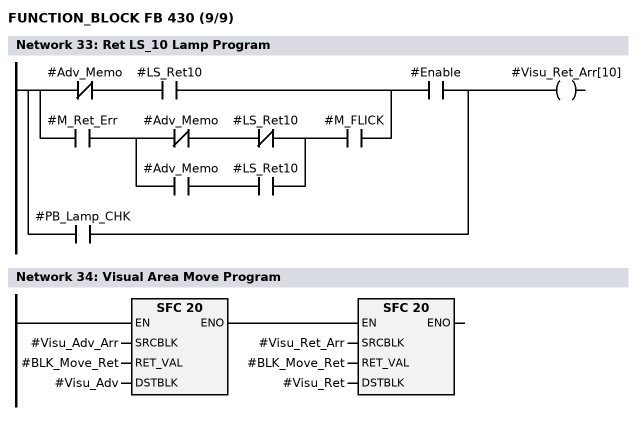
      A(    ;
      AN    #Adv_Memo;
      A     #LS_Ret10;
      O     ;
      A     #M_Ret_Err;
      A(    ;
      AN    #Adv_Memo;
      AN    #LS_Ret10;
      O     ;
      A     #Adv_Memo;
      A     #LS_Ret10;
      )     ;
      A     #M_FLICK;
      )     ;
      A     #Enable;
      O     #PB_Lamp_CHK;
      =     #Visu_Ret_Arr[10];
NETWORK
TITLE =Visual Area Move Program

      A(    ;
      CALL SFC   20 (
           SRCBLK                   := #Visu_Adv_Arr,
           RET_VAL                  := #BLK_Move_Ret,
           DSTBLK                   := #Visu_Adv);
      A     BR;
      )     ;
      JNB   _001;
      CALL SFC   20 (
           SRCBLK                   := #Visu_Ret_Arr,
           RET_VAL                  := #BLK_Move_Ret,
           DSTBLK                   := #Visu_Ret);
_001: NOP   0;
END_FUNCTION_BLOCK

FUNCTION_BLOCK FB 470
TITLE =HMI Body Type Modify Variables Program
AUTHOR : HMC
FAMILY : HMI
NAME : HMI
VERSION : 1.0


VAR_INPUT
  Station : INT ;
  HMI_Disp_DB : INT ;
  HMI_Disp_Add : INT ;
  CType_DB : INT ;
  CType_Start_Add : INT ;
  Byte_per_Stn : INT ;
  M_Modify_OK : BOOL ;
  SS_CCR_On : BOOL ;
  PB_Set : BOOL ;
  PB_Reset : BOOL ;
END_VAR
VAR_OUTPUT
  LP_CCR_On : BOOL ;
  LP_Modify_On : BOOL ;
END_VAR
VAR
  Source_Data : WORD ;
  Modify_Data : WORD ;
  Pre_Station : INT ;
  Station_PLS : BOOL ;
  Source_Add : INT ;
  SFC20_Ret : INT ;
  Fill_Source : WORD ;
END_VAR
VAR_TEMP
  Source_Area : ANY ;
  Modify_Area : ANY ;
END_VAR
BEGIN
NETWORK
TITLE =FAC On Lamp Program

      A     #SS_CCR_On;
      =     #LP_CCR_On;
NETWORK
TITLE =Operation Pulse

      L     #Station; // Station Select Data
      L     0; // Is Not Zero
      <>I   ;
      JNB   _End; // Jump to End
NETWORK
TITLE =Modify On Lamp Program
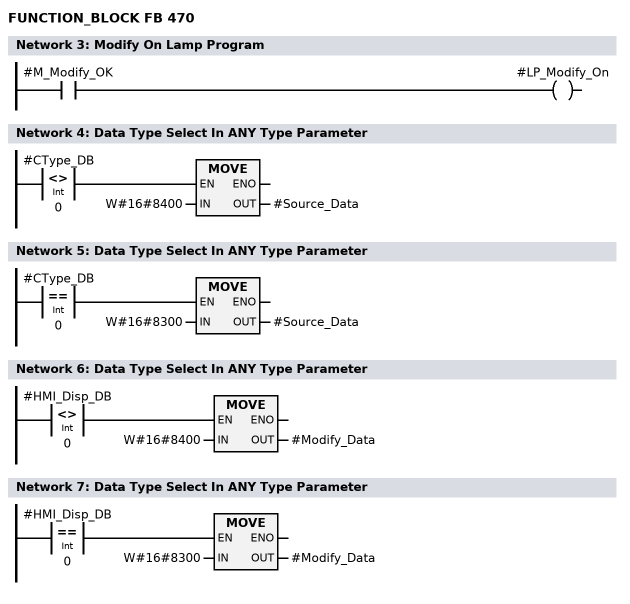

      A     #M_Modify_OK;
      =     #LP_Modify_On;
NETWORK
TITLE =Data Type Select In ANY Type Parameter

      A(    ; // If Source DB is Not Zero
      L     #CType_DB;
      L     0;
      <>I   ;
      )     ;
      JNB   _B01; // Jump to Next Step
      L     W#16#8400; // Load "8400" _ Means "DB Area"
      T     #Source_Data; // Transfer to Data_Type
_B01: NOP   0;
NETWORK
TITLE =Data Type Select In ANY Type Parameter

      A(    ; // If DB_NO is Zero
      L     #CType_DB;
      L     0;
      ==I   ;
      )     ;
      JNB   _B02; // Jump to Next Step
      L     W#16#8300; // Load "8300" _ Means "Bit Memory Area"
      T     #Source_Data; // Transfer to Data_Type
_B02: NOP   0;
NETWORK
TITLE =Data Type Select In ANY Type Parameter

      A(    ; // If Source DB is Not Zero
      L     #HMI_Disp_DB;
      L     0;
      <>I   ;
      )     ;
      JNB   _B03; // Jump to Next Step
      L     W#16#8400; // Load "8400" _ Means "DB Area"
      T     #Modify_Data; // Transfer to Data_Type
_B03: NOP   0;
NETWORK
TITLE =Data Type Select In ANY Type Parameter

      A(    ; // If DB_NO is Zero
      L     #HMI_Disp_DB;
      L     0;
      ==I   ;
      )     ;
      JNB   _B04; // Jump to Next Step
      L     W#16#8300; // Load "8300" _ Means "Bit Memory Area"
      T     #Modify_Data; // Transfer to Data_Type
_B04: NOP   0;
NETWORK
TITLE =Source Area Start Address Calculate Porgram

      L     #Station; // Station Amount - 1
      L     1;
      -I    ;
      L     #Byte_per_Stn; // Multi Length Per Station
      *I    ;
      L     #CType_Start_Add;
      +I    ;
      T     #Source_Add;
NETWORK
TITLE =Make a "ANY" Type Data

      LAR1  P##Source_Area; // Load 1st Station Address of ANY Pointer In "AR1"

      L     B#16#10; // Load Syntax ID For S7 "10"
      T     LB [AR1,P#0.0]; // Transfer ID to the ANY Pointer

      L     B#16#2; // Load Data Type _ "2" means "BYTE"
      T     LB [AR1,P#1.0]; // Transfer Data Type to the ANY Pointer

      L     #Byte_per_Stn; // Load the Length of Source Data
      T     LW [AR1,P#2.0]; // Transfer the Numbers to the ANY Pointer

      L     #CType_DB; // Load DB Number _ "0" means don't use "DB"
      T     LW [AR1,P#4.0]; // Transfer the Numbers to the ANY Pointer

      L     #Source_Data; // Load Data Type _ "83" means "Bit Memory" Area
      T     LW [AR1,P#6.0]; //                  "84" means "DB" Area

      L     #Source_Add; // Load Start Address
      SLW   3; // Shift Left Word _ "3" Bit
      T     LW [AR1,P#8.0]; // Transfer the Address to the ANY Pointer

      LAR1  P##Modify_Area; // Load 2nd Station Address of ANY Pointer In "AR1"

      L     B#16#10; //Load Syntax ID For S7 "10"
      T     LB [AR1,P#0.0]; //Load Syntax ID For S7 "10"

      L     B#16#2; //  Load Data Type _ "2" means "BYTE"
      T     LB [AR1,P#1.0]; // Transfer Data Type to the ANY Pointer

      L     #Byte_per_Stn; // Load the Length of Target Data
      T     LW [AR1,P#2.0]; // Transfer the Numbers to the ANY Pointer

      L     #HMI_Disp_DB; // Load DB Number _ "0" means don't use "DB"
      T     LW [AR1,P#4.0]; // Transfer the Numbers to the ANY Pointer

      L     #Modify_Data; // Load Data Type _ "83" means "Bit Memory" Area
      T     LW [AR1,P#6.0]; //                  "84" means "DB" Area

      L     #HMI_Disp_Add; //  Load Start Address
      SLW   3; // Shift Left Word _ "3" Bit
      T     LW [AR1,P#8.0]; // Transfer the Address to the ANY Pointer

NETWORK
TITLE =Copy To Modify Area Program

      L     #Station;
      L     #Pre_Station;
      <>I   ;
      JNB   _B05;
NETWORK
TITLE =Copy To Previous Station No Program

      L     #Station;
      T     #Pre_Station;
NETWORK
TITLE =Block Move to Modify Area


      CALL SFC   20 (
           SRCBLK                   := #Source_Area,
           RET_VAL                  := #SFC20_Ret,
           DSTBLK                   := #Modify_Area);
_B05: NOP   0;
NETWORK
TITLE =Data Clear Program

      A     #M_Modify_OK;
      A     #PB_Reset;
      JNB   _B06;
NETWORK
TITLE =Clear Source Data Area


      CALL SFC   21 (
           BVAL                     := #Fill_Source,// "Zero"
           RET_VAL                  := #SFC20_Ret,
           BLK                      := #Source_Area);// Transfer to First Station Area

NETWORK
TITLE =Clear Source Data Area


      CALL SFC   21 (
           BVAL                     := #Fill_Source,// "Zero"
           RET_VAL                  := #SFC20_Ret,
           BLK                      := #Modify_Area);// Transfer to First Station Area
_B06: NOP   0;
NETWORK
TITLE =Data Clear Program

      A     #M_Modify_OK;
      A     #PB_Set;
      JNB   _B07;
NETWORK
TITLE =Block Move to Modify Area


      CALL SFC   20 (
           SRCBLK                   := #Modify_Area,
           RET_VAL                  := #SFC20_Ret,
           DSTBLK                   := #Source_Area);
_B07: NOP   0;
NETWORK
TITLE =


_End: NOP   0;

END_FUNCTION_BLOCK

FUNCTION FC 502 : VOID
TITLE =
VERSION : 1.0


VAR_INPUT
  FAC_Log_DB_NO : INT ;	//FAC Log 저장용 DB번호
  LOG_INDEX : WORD ;	//Log저장용 Data의 Index값
  LOG_DEC_DATA : INT ;	//Log저장용 Data의 현재 상태값
  LOG_BCD_DATA : WORD ;	//Log저장용 Data의 VIN No4
END_VAR
VAR_TEMP
  FAC_Log_DB : INT ;	//FAC Log 저장용 DB번호 Temp
  DATE_TIME : DATE_AND_TIME ;	//System Date&Time
  READ_CLK_VAR : INT ;	//System Date&Time 읽기 실행 Return값
END_VAR
BEGIN
NETWORK
TITLE =FAC Log 저장용 DB Open


      L     #FAC_Log_DB_NO;
      T     #FAC_Log_DB;
      OPN   DB [#FAC_Log_DB];

      L     0;
      T     DBW   92;
      NOP   0;
NETWORK
TITLE =Log Data Shift실행용 최초 Byte 위치 설정



      A(    ;
      L     1090;
      T     DBW   94;
      SET   ;
      SAVE  ;
      CLR   ;
      A     BR;
      )     ;
      JNB   _001;
      L     DBW   94;
      L     10;
      -I    ;
      T     DBW   96;
_001: NOP   0;


NETWORK
TITLE =Log Data Shift실행용 LOOP(99회)

a:    L     100;
      L     DBW   92;
      ==I   ;
      JC    END;

      L     DBW   94; //132
      SLW   3;
      LAR1  ;

      L     DBW   96; //132
      SLW   3;
      LAR2  ;

      L     DBD [AR2,P#0.0];
      T     DBD [AR1,P#0.0];
      L     DBD [AR2,P#4.0];
      T     DBD [AR1,P#4.0];
      L     DBW [AR2,P#8.0];
      T     DBW [AR1,P#8.0];

      L     DBW   94;
      L     10;
      -I    ;
      T     DBW   94;

      L     DBW   96;
      L     10;
      -I    ;
      T     DBW   96;

      L     1;
      L     DBW   92;
      +I    ;
      T     DBW   92;
      JP    a;
END:  NOP   0;
      LAR1  P#0.0;

NETWORK
TITLE =System Date & Time 읽기용 시스템 함수 호출

      CALL SFC    1 (
           RET_VAL                  := #READ_CLK_VAR,
           CDT                      := #DATE_TIME);
      NOP   0;


NETWORK
TITLE =현재 발생한 정보에 대한 Log저장

      LAR2  P#0.0;
      L     #LOG_INDEX;
      T     DBW [AR1,P#100.0];

      LAR1  P##DATE_TIME;
      L     LB [AR1,P#2.0];
      T     DBB [AR2,P#102.0];
      L     LB [AR1,P#3.0];
      T     DBB [AR2,P#103.0];
      L     LB [AR1,P#4.0];
      T     DBB [AR2,P#104.0];
      L     LB [AR1,P#5.0];
      T     DBB [AR2,P#105.0];

      L     #LOG_DEC_DATA;
      T     DBW [AR2,P#106.0];
      L     #LOG_BCD_DATA;
      T     DBW [AR2,P#108.0];

      NOP   0;

END_FUNCTION

FUNCTION FC 503 : VOID
TITLE =
VERSION : 0.1


VAR_INPUT
  Data_DB : INT ;
  Data_Length : INT ;
  FillStart_Add : INT ;
  Fill_Data : BYTE ;
END_VAR
VAR_TEMP
  Source_DB : ANY ;
  Data_DB_temp : INT ;
  Data_Length_temp : INT ;
  FillStart_Add_temp : INT ;
  Fill_Data_temp : BYTE ;
  Rcv_Val : INT ;
END_VAR
BEGIN
NETWORK
TITLE =

      L     #Data_DB;
      T     #Data_DB_temp;
      L     #Data_Length;
      T     #Data_Length_temp;
      L     #FillStart_Add;
      T     #FillStart_Add_temp;
      L     #Fill_Data;
      T     #Fill_Data_temp;

      OPN   DB [#Data_DB_temp];
//      LAR1  P#0.0


      LAR1  P##Source_DB;
      L     B#16#10;
      T     LB [AR1,P#0.0]; //S7 Defualt
      L     B#16#2;
      T     LB [AR1,P#1.0]; //Data Type 'Byte'
      L     #Data_Length_temp;
      T     LW [AR1,P#2.0]; //Send Counter
      L     #Data_DB_temp;
      T     LW [AR1,P#4.0]; //DB_No. Set
      L     W#16#8400;
      T     LW [AR1,P#6.0]; //Area Select
      L     #FillStart_Add_temp;
      SLW   3;
      T     LW [AR1,P#8.0]; //Byte.Bit Address Set


      CALL SFC   21 (
           BVAL                     := #Fill_Data_temp,
           RET_VAL                  := #Rcv_Val,
           BLK                      := #Source_DB);


      NOP   0;
END_FUNCTION

FUNCTION FC 504 : VOID
TITLE =
VERSION : 0.1


VAR_INPUT
  SourceData_DB : INT ;
  SourceStart_Add : INT ;
  BLKMOV_Byte_Length : INT ;
  DestData_DB : INT ;
  DestStart_Add : INT ;
END_VAR
VAR_TEMP
  Source_DB : ANY ;
  Dest_DB : ANY ;
  SourceData_DB_temp : INT ;
  BLKMOV_Byte_Length_temp : INT ;
  SourceStart_Add_temp : INT ;
  DestData_DB_Temp : INT ;
  DestStart_Add_Temp : INT ;
  Send_Val : INT ;
END_VAR
BEGIN
NETWORK
TITLE =

      L     #SourceData_DB;
      T     #SourceData_DB_temp;

      L     #BLKMOV_Byte_Length;
      T     #BLKMOV_Byte_Length_temp;

      L     #SourceStart_Add;
      T     #SourceStart_Add_temp;

      L     #DestData_DB;
      T     #DestData_DB_Temp;

      L     #DestStart_Add;
      T     #DestStart_Add_Temp;


      OPN   DB [#SourceData_DB_temp];

      LAR1  P##Source_DB;
      L     B#16#10;
      T     LB [AR1,P#0.0]; //S7 Defualt
      L     B#16#2;
      T     LB [AR1,P#1.0]; //Data Type 'Byte'
      L     #BLKMOV_Byte_Length_temp;
      T     LW [AR1,P#2.0]; //Send Counter
      L     #SourceData_DB_temp;
      T     LW [AR1,P#4.0]; //DB_No. Set
      L     W#16#8400;
      T     LW [AR1,P#6.0]; //Area Select
      L     #SourceStart_Add_temp;
      SLW   3;
      T     LW [AR1,P#8.0]; //Byte.Bit Address Set


      LAR2  P##Dest_DB;
      L     B#16#10;
      T     LB [AR2,P#0.0]; //S7 Defualt
      L     B#16#2;
      T     LB [AR2,P#1.0]; //Data Type 'Byte'
      L     #BLKMOV_Byte_Length;
      T     LW [AR2,P#2.0]; //Recieve Counter
      L     #DestData_DB_Temp;
      T     LW [AR2,P#4.0]; //DB_No. Set
      L     W#16#8400;
      T     LW [AR2,P#6.0]; //Area Select
      L     #DestStart_Add_Temp;
      SLW   3;
      T     LW [AR2,P#8.0]; //Byte.Bit Address Set



      CALL SFC   20 (
           SRCBLK                   := #Source_DB,
           RET_VAL                  := #Send_Val,
           DSTBLK                   := #Dest_DB);

      NOP   0;
END_FUNCTION

FUNCTION FC 505 : VOID
TITLE =
VERSION : 0.1


VAR_INPUT
  FAC_DB : INT ;
  FAC_LOG_DB : INT ;
END_VAR
VAR_TEMP
  FAC_DB_NO : INT ;
  FAC_LOG_DB_NO : INT ;
  Read_DATE_TIME : DATE_AND_TIME ;
  Set_DATE_TIME : DATE_AND_TIME ;
  READ_CLK_VAR : INT ;
  Set_CLK_VAR : INT ;
  Set_CLK_ON : BOOL ;
END_VAR
BEGIN
NETWORK
TITLE =System Date & Time 읽기용 시스템 함수 호출

      L     #FAC_LOG_DB;
      T     #FAC_LOG_DB_NO;
      L     #FAC_DB;
      T     #FAC_DB_NO;
      OPN   DB [#FAC_DB_NO];
      OPN   DI [#FAC_LOG_DB_NO];

      LAR1  P#0.0;
      LAR2  P#0.0;

NETWORK
TITLE =System Date & Time 읽기용 시스템 함수 호출

      CALL SFC    1 (
           RET_VAL                  := #READ_CLK_VAR,
           CDT                      := #Read_DATE_TIME);
      NOP   0;
NETWORK
TITLE =현재 발생한 정보에 대한 Log저장


      LAR1  P#0.0;
      LAR2  P#0.0;

      LAR1  P##Read_DATE_TIME;
      L     LB [AR1,P#0.0];
      T     DIB [AR2,P#40.0];
      L     LB [AR1,P#1.0];
      T     DIB [AR2,P#41.0];


      NOP   0;

NETWORK
TITLE =

      LAR1  P#0.0;
      LAR2  P#0.0;

      LAR2  P##Set_DATE_TIME;
      L     DIB [AR1,P#40.0];
      T     LB [AR2,P#0.0];
      L     DIB [AR1,P#41.0];
      T     LB [AR2,P#1.0];
      L     DBB  962;
      T     LB [AR2,P#2.0];
      L     DBB  963;
      T     LB [AR2,P#3.0];
      L     DBB  960;
      T     LB [AR2,P#4.0];
      L     DBB  961;
      T     LB [AR2,P#5.0];
      NOP   0;
NETWORK
TITLE =
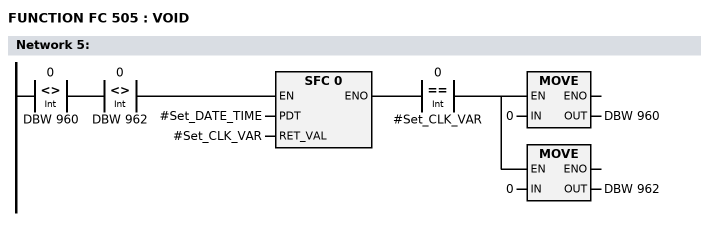

      A(    ;
      A(    ;
      L     0;
      L     DBW  960;
      <>I   ;
      )     ;
      A(    ;
      L     0;
      L     DBW  962;
      <>I   ;
      )     ;
      JNB   _001;
      CALL SFC    0 (
           PDT                      := #Set_DATE_TIME,
           RET_VAL                  := #Set_CLK_VAR);
_001: A     BR;
      )     ;
      A(    ;
      L     0;
      L     #Set_CLK_VAR;
      ==I   ;
      )     ;
      =     L     25.0;
      A     L     25.0;
      JNB   _002;
      L     0;
      T     DBW  960;
_002: NOP   0;
      A     L     25.0;
      JNB   _003;
      L     0;
      T     DBW  962;
_003: NOP   0;
END_FUNCTION

FUNCTION_BLOCK FB 512
TITLE =Car Type Variables Program
AUTHOR : HMC
FAMILY : Car_Type
NAME : Car_Type
VERSION : 1.0


VAR_INPUT
  Stn_Vin_No : DINT ;	//Startadress Inputs from HW-Konfig
  Stn_Bt_1Word : WORD ;
  Stn_Bt_2Word : WORD ;
  Stn_Bt_3Word : WORD ;
  Stn_Bt_4Word : WORD ;
  Stn_Bt_5Word_Sp : WORD ;
  Stn_Bt_6Word_Sp : WORD ;
END_VAR
VAR_OUTPUT
  M_BType_On : BOOL ;
  M_BType_None : BOOL ;
  M_Bypass_BType : BOOL ;
  M_BType_TL : BOOL ;
  M_BType_LM : BOOL ;
  M_BType_SP1 : BOOL ;
  M_BType_SP2 : BOOL ;
  M_BType_SP3 : BOOL ;
  M_BType_DOM : BOOL ;
  M_BType_EXP : BOOL ;
  Robot_Prog_No : INT ;
END_VAR
VAR
  STN_Btype_1Arr : ARRAY  [0 .. 15 ] OF BOOL ;
  STN_Btype_2Arr : ARRAY  [0 .. 15 ] OF BOOL ;
  STN_Btype_3Arr : ARRAY  [0 .. 15 ] OF BOOL ;
  STN_Btype_4Arr : ARRAY  [0 .. 15 ] OF BOOL ;
  STN_Btype_5Arr : ARRAY  [0 .. 15 ] OF BOOL ;
  STN_Btype_6Arr : ARRAY  [0 .. 15 ] OF BOOL ;
  STN_1st_BT_On : BOOL ;
  STN_2nd_BT_On : BOOL ;
  STN_3rd_BT_On : BOOL ;
  STN_4th_BT_On : BOOL ;
  STN_5th_BT_On : BOOL ;
  STN_6th_BT_On : BOOL ;
  STN_7th_BT_On : BOOL ;
  STN_8th_BT_On : BOOL ;
  STN_9th_BT_On : BOOL ;
  STN_10th_BT_On : BOOL ;
  STN_11th_BT_On : BOOL ;
  STN_12th_BT_On : BOOL ;
  STN_1st_BT_Off : BOOL ;
  BLKMove_Ret : INT ;
  VIN_1BCD : WORD ;
  VIN_2BCD : WORD ;
  VIN_1Int : INT ;
  VIN_2Int : INT ;
END_VAR
BEGIN
NETWORK
TITLE =Station Body Type Data Change to 16-bit array

      CALL SFC   20 (
           SRCBLK                   := #Stn_Bt_1Word,
           RET_VAL                  := #BLKMove_Ret,
           DSTBLK                   := #STN_Btype_1Arr);
      NOP   0;
NETWORK
TITLE =Station Body Type Data Change to 16-bit array

      CALL SFC   20 (
           SRCBLK                   := #Stn_Bt_2Word,
           RET_VAL                  := #BLKMove_Ret,
           DSTBLK                   := #STN_Btype_2Arr);
      NOP   0;
NETWORK
TITLE =Station Body Type Data Change to 16-bit array

      CALL SFC   20 (
           SRCBLK                   := #Stn_Bt_3Word,
           RET_VAL                  := #BLKMove_Ret,
           DSTBLK                   := #STN_Btype_3Arr);
      NOP   0;
NETWORK
TITLE =Station Body Type Data Change to 16-bit array

      CALL SFC   20 (
           SRCBLK                   := #Stn_Bt_4Word,
           RET_VAL                  := #BLKMove_Ret,
           DSTBLK                   := #STN_Btype_4Arr);
      NOP   0;
NETWORK
TITLE =Station Body Type Data Change to 16-bit array

      CALL SFC   20 (
           SRCBLK                   := #Stn_Bt_5Word_Sp,
           RET_VAL                  := #BLKMove_Ret,
           DSTBLK                   := #STN_Btype_5Arr);
      NOP   0;
NETWORK
TITLE =Station Body Type Data Change to 16-bit array

      CALL SFC   20 (
           SRCBLK                   := #Stn_Bt_6Word_Sp,
           RET_VAL                  := #BLKMove_Ret,
           DSTBLK                   := #STN_Btype_6Arr);
      NOP   0;
NETWORK
TITLE =공정 1차종

      AN    OV;
      A(    ;
      O     #STN_Btype_1Arr[0];
      O     #STN_Btype_1Arr[1];
      O     #STN_Btype_1Arr[2];
      O     #STN_Btype_1Arr[3];
      O     #STN_Btype_1Arr[4];
      )     ;
      =     #STN_1st_BT_On;
NETWORK
TITLE =공정 2차종

      AN    OV;
      A(    ;
      O     #STN_Btype_1Arr[5];
      O     #STN_Btype_1Arr[6];
      O     #STN_Btype_1Arr[7];
      O     #STN_Btype_1Arr[8];
      )     ;
      =     #STN_2nd_BT_On;
NETWORK
TITLE =공정 3차종

      AN    OV;
      A(    ;
      O     #STN_Btype_1Arr[9];
      O     #STN_Btype_1Arr[10];
      )     ;
      =     #STN_3rd_BT_On;
NETWORK
TITLE =공정 4차종

      AN    OV;
      A(    ;
      O     #STN_Btype_1Arr[11];
      O     #STN_Btype_1Arr[12];
      O     #STN_Btype_1Arr[13];
      O     #STN_Btype_1Arr[14];
      O     #STN_Btype_1Arr[15];
      O     #STN_Btype_2Arr[0];
      O     #STN_Btype_2Arr[1];
      O     #STN_Btype_2Arr[2];
      O     #STN_Btype_2Arr[3];
      O     #STN_Btype_2Arr[4];
      O     #STN_Btype_2Arr[5];
      )     ;
      =     #STN_4th_BT_On;
NETWORK
TITLE =공정 5차종

      AN    OV;
      A(    ;
      O     #STN_Btype_2Arr[6];
      O     #STN_Btype_2Arr[7];
      )     ;
      =     #STN_5th_BT_On;
NETWORK
TITLE =공정 6차종

      AN    OV;
      A(    ;
      O     #STN_Btype_2Arr[8];
      O     #STN_Btype_2Arr[9];
      O     #STN_Btype_2Arr[10];
      O     #STN_Btype_2Arr[11];
      O     #STN_Btype_2Arr[12];
      O     #STN_Btype_2Arr[13];
      O     #STN_Btype_2Arr[14];
      O     #STN_Btype_2Arr[15];
      )     ;
      =     #STN_6th_BT_On;
NETWORK
TITLE =공정 7차종

      AN    OV;
      A(    ;
      O     #STN_Btype_3Arr[0];
      O     #STN_Btype_3Arr[1];
      )     ;
      =     #STN_7th_BT_On;
NETWORK
TITLE =공정 8차종

      AN    OV;
      A(    ;
      O     #STN_Btype_3Arr[2];
      O     #STN_Btype_3Arr[3];
      O     #STN_Btype_3Arr[6];
      )     ;
      =     #STN_8th_BT_On;
NETWORK
TITLE =공정 9차종

      AN    OV;
      A(    ;
      O     #STN_Btype_3Arr[4];
      O     #STN_Btype_3Arr[5];
      )     ;
      =     #STN_9th_BT_On;
NETWORK
TITLE =공정 10차종

      AN    OV;
      A(    ;
      O     #STN_Btype_3Arr[6];
      O     #STN_Btype_3Arr[7];
      ON    #STN_10th_BT_On;
      )     ;
      =     #STN_10th_BT_On;
NETWORK
TITLE =공정 11차종

      AN    OV;
      A(    ;
      O     #STN_Btype_3Arr[8];
      O     #STN_Btype_3Arr[9];
      O     #STN_Btype_3Arr[10];
      O     #STN_Btype_3Arr[11];
      O     #STN_Btype_3Arr[12];
      O     #STN_Btype_3Arr[13];
      O     #STN_Btype_3Arr[14];
      O     #STN_Btype_3Arr[15];
      O     #STN_Btype_4Arr[0];
      O     #STN_Btype_4Arr[1];
      O     #STN_Btype_4Arr[2];
      O     #STN_Btype_4Arr[3];
      O     #STN_Btype_4Arr[4];
      O     #STN_Btype_4Arr[5];
      O     #STN_Btype_4Arr[6];
      O     #STN_Btype_4Arr[7];
      O     #STN_Btype_4Arr[8];
      O     #STN_Btype_4Arr[9];
      )     ;
      =     #STN_11th_BT_On;
NETWORK
TITLE =공정 차종 있음
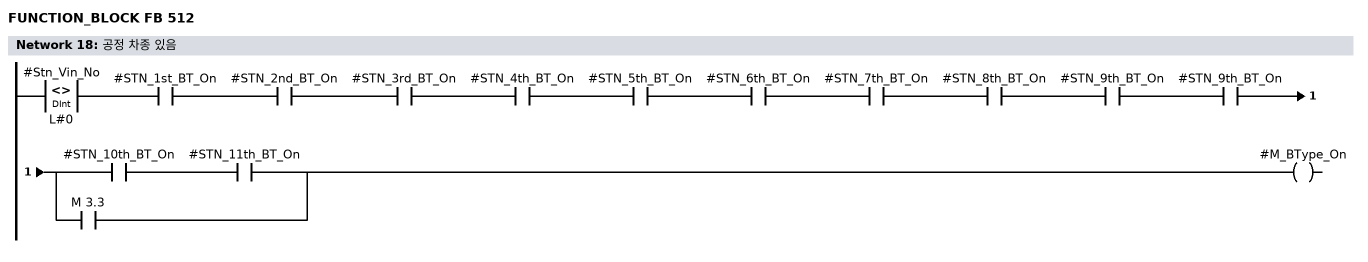

      A(    ;
      L     #Stn_Vin_No;
      L     L#0;
      <>D   ;
      )     ;
      A     #STN_1st_BT_On;
      A     #STN_2nd_BT_On;
      A     #STN_3rd_BT_On;
      A     #STN_4th_BT_On;
      A     #STN_5th_BT_On;
      A     #STN_6th_BT_On;
      A     #STN_7th_BT_On;
      A     #STN_8th_BT_On;
      A     #STN_9th_BT_On;
      A     #STN_9th_BT_On;
      A(    ;
      A     #STN_10th_BT_On;
      A     #STN_11th_BT_On;
      O     M      3.3;
      )     ;
      =     #M_BType_On;
NETWORK
TITLE =1차종 없음

      AN    OV;
      AN    #STN_Btype_1Arr[0];
      AN    #STN_Btype_1Arr[1];
      AN    #STN_Btype_1Arr[2];
      AN    #STN_Btype_1Arr[3];
      AN    #STN_Btype_1Arr[4];
      =     #STN_1st_BT_Off;
NETWORK
TITLE =공정 차종 없음
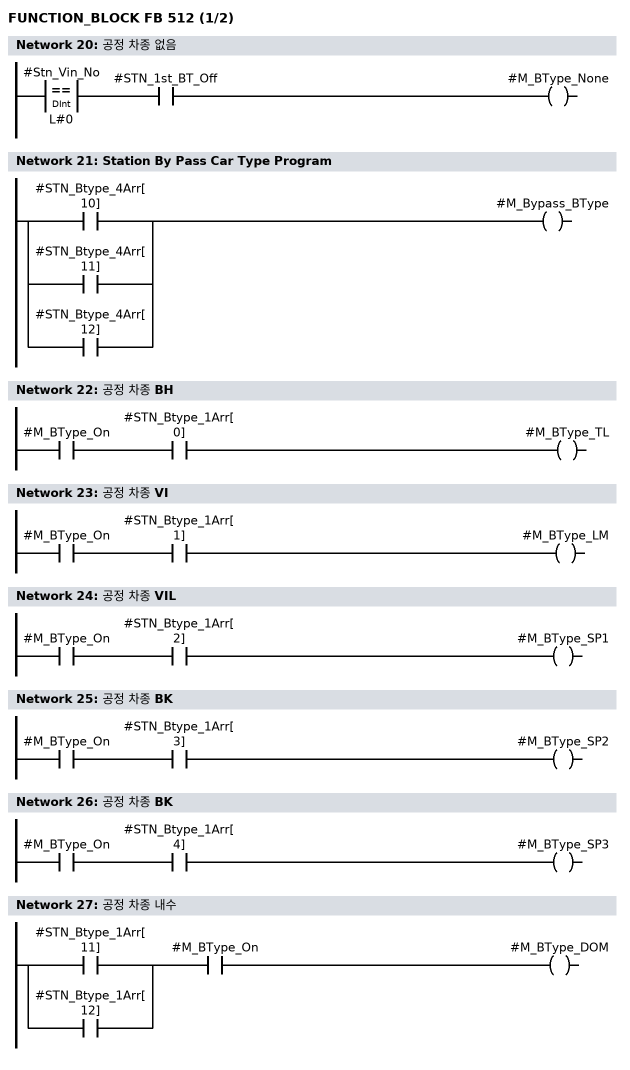

      A(    ;
      L     #Stn_Vin_No;
      L     L#0;
      ==D   ;
      )     ;
      A     #STN_1st_BT_Off;
      =     #M_BType_None;
NETWORK
TITLE =Station By Pass Car Type Program

      O     #STN_Btype_4Arr[10];
      O     #STN_Btype_4Arr[11];
      O     #STN_Btype_4Arr[12];
      =     #M_Bypass_BType;
NETWORK
TITLE =공정 차종 BH

      A     #M_BType_On;
      A     #STN_Btype_1Arr[0];
      =     #M_BType_TL;
NETWORK
TITLE =공정 차종 VI

      A     #M_BType_On;
      A     #STN_Btype_1Arr[1];
      =     #M_BType_LM;
NETWORK
TITLE =공정 차종 VIL

      A     #M_BType_On;
      A     #STN_Btype_1Arr[2];
      =     #M_BType_SP1;
NETWORK
TITLE =공정 차종 BK

      A     #M_BType_On;
      A     #STN_Btype_1Arr[3];
      =     #M_BType_SP2;
NETWORK
TITLE =공정 차종 BK

      A     #M_BType_On;
      A     #STN_Btype_1Arr[4];
      =     #M_BType_SP3;
NETWORK
TITLE =공정 차종 내수

      A(    ;
      O     #STN_Btype_1Arr[11];
      O     #STN_Btype_1Arr[12];
      )     ;
      A     #M_BType_On;
      =     #M_BType_DOM;
NETWORK
TITLE =공정 차종 수출
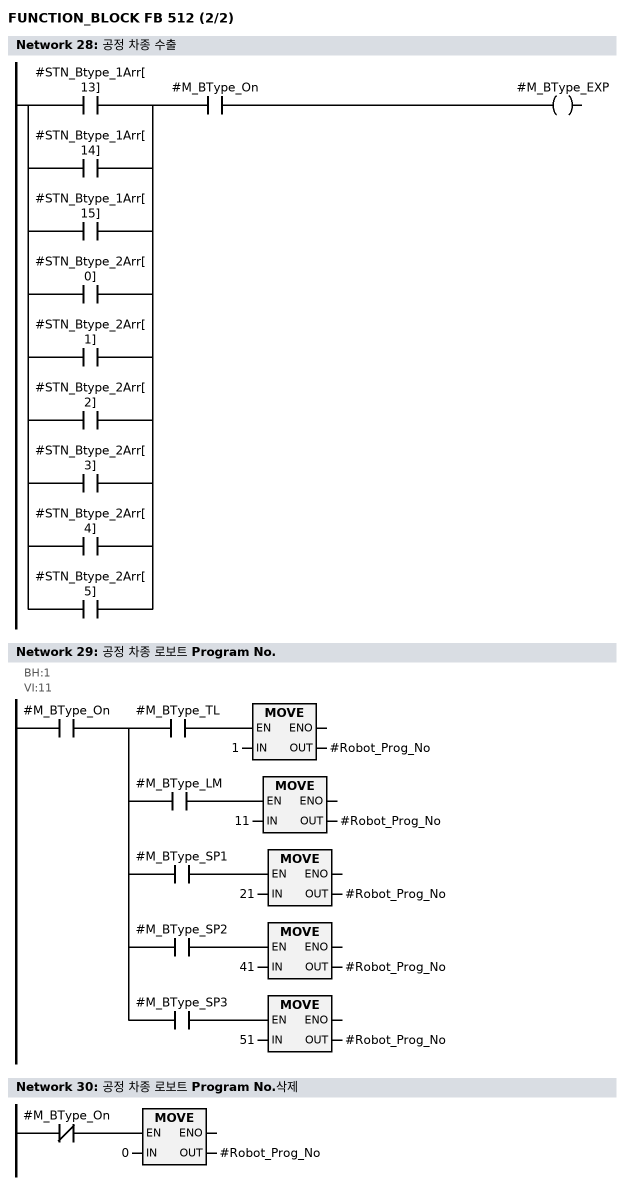

      A(    ;
      O     #STN_Btype_1Arr[13];
      O     #STN_Btype_1Arr[14];
      O     #STN_Btype_1Arr[15];
      O     #STN_Btype_2Arr[0];
      O     #STN_Btype_2Arr[1];
      O     #STN_Btype_2Arr[2];
      O     #STN_Btype_2Arr[3];
      O     #STN_Btype_2Arr[4];
      O     #STN_Btype_2Arr[5];
      )     ;
      A     #M_BType_On;
      =     #M_BType_EXP;
NETWORK
TITLE =공정 차종 로보트 Program No.
//BH:1
//VI:11
      A     #M_BType_On;
      =     L      0.0;
      A     L      0.0;
      A     #M_BType_TL;
      JNB   _001;
      L     1;
      T     #Robot_Prog_No;
_001: NOP   0;
      A     L      0.0;
      A     #M_BType_LM;
      JNB   _002;
      L     11;
      T     #Robot_Prog_No;
_002: NOP   0;
      A     L      0.0;
      A     #M_BType_SP1;
      JNB   _003;
      L     21;
      T     #Robot_Prog_No;
_003: NOP   0;
      A     L      0.0;
      A     #M_BType_SP2;
      JNB   _004;
      L     41;
      T     #Robot_Prog_No;
_004: NOP   0;
      A     L      0.0;
      A     #M_BType_SP3;
      JNB   _005;
      L     51;
      T     #Robot_Prog_No;
_005: NOP   0;
NETWORK
TITLE =공정 차종 로보트 Program No.삭제

      AN    #M_BType_On;
      JNB   _006;
      L     0;
      T     #Robot_Prog_No;
_006: NOP   0;
END_FUNCTION_BLOCK

FUNCTION FC 98 : VOID
TITLE =
VERSION : 0.1


VAR_TEMP
  SFC20_RET_VAL : INT ;
  RECV1_LEN : WORD ;
  SEND1_LEN : WORD ;
  RECV2_LEN : WORD ;
  SEND2_LEN : WORD ;
  RECV3_LEN : WORD ;
  SEND3_LEN : WORD ;
END_VAR
BEGIN
NETWORK
TITLE =
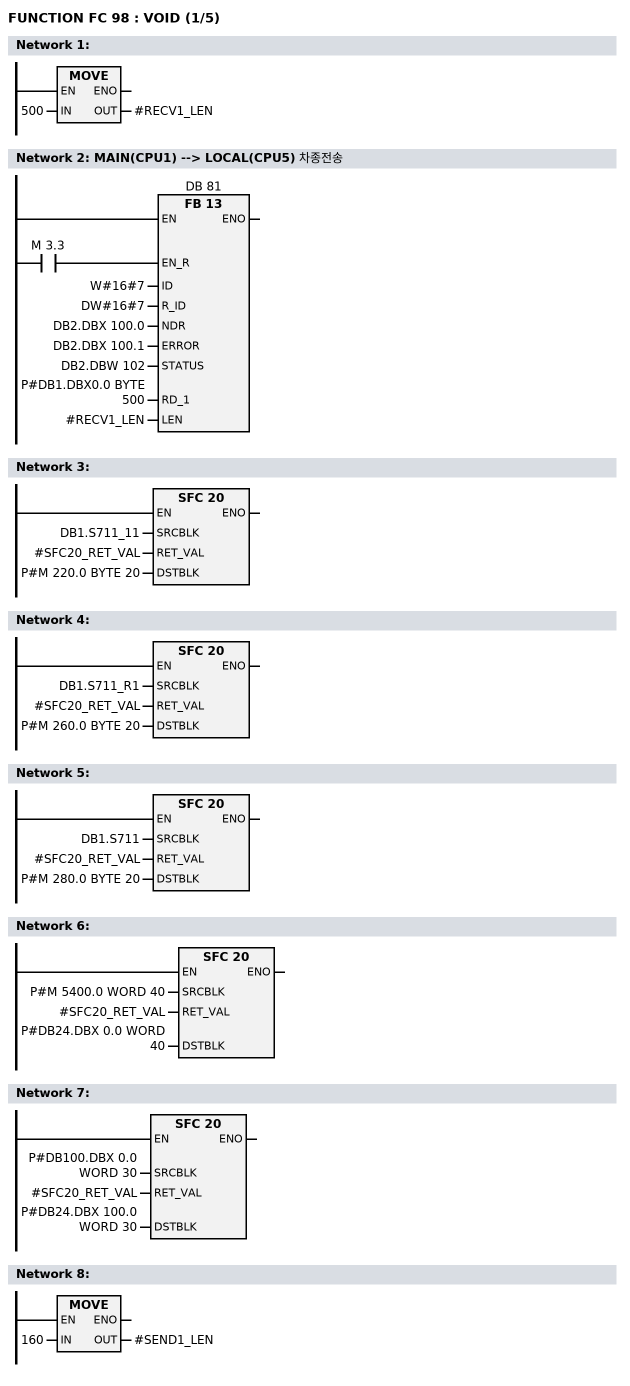

      L     500;
      T     #RECV1_LEN;
      NOP   0;
NETWORK
TITLE =MAIN(CPU1) --> LOCAL(CPU5) 차종전송

      A     M      3.3;
      =     L     14.0;
      BLD   103;
      CALL FB    13 , DB    81 (
           EN_R                     := L     14.0,
           ID                       := W#16#7,
           R_ID                     := DW#16#7,
           NDR                      := DB2.DBX  100.0,
           ERROR                    := DB2.DBX  100.1,
           STATUS                   := DB2.DBW  102,
           RD_1                     := P#DB1.DBX0.0 BYTE 500,
           LEN                      := #RECV1_LEN);
      NOP   0;
NETWORK
TITLE =

      CALL SFC   20 (
           SRCBLK                   := DB1.S711_11,
           RET_VAL                  := #SFC20_RET_VAL,
           DSTBLK                   := P#M 220.0 BYTE 20);
      NOP   0;
NETWORK
TITLE =

      CALL SFC   20 (
           SRCBLK                   := DB1.S711_R1,
           RET_VAL                  := #SFC20_RET_VAL,
           DSTBLK                   := P#M 260.0 BYTE 20);
      NOP   0;
NETWORK
TITLE =

      CALL SFC   20 (
           SRCBLK                   := DB1.S711,
           RET_VAL                  := #SFC20_RET_VAL,
           DSTBLK                   := P#M 280.0 BYTE 20);
      NOP   0;
NETWORK
TITLE =

      CALL SFC   20 (
           SRCBLK                   := P#M 5400.0 WORD 40,
           RET_VAL                  := #SFC20_RET_VAL,
           DSTBLK                   := P#DB24.DBX 0.0 WORD 40);
      NOP   0;
NETWORK
TITLE =

      CALL SFC   20 (
           SRCBLK                   := P#DB100.DBX 0.0 WORD 30,
           RET_VAL                  := #SFC20_RET_VAL,
           DSTBLK                   := P#DB24.DBX 100.0 WORD 30);
      NOP   0;
NETWORK
TITLE =

      L     160;
      T     #SEND1_LEN;
      NOP   0;
NETWORK
TITLE =LOCAL(CPU5) --> MAIN(CPU1) 공정상태
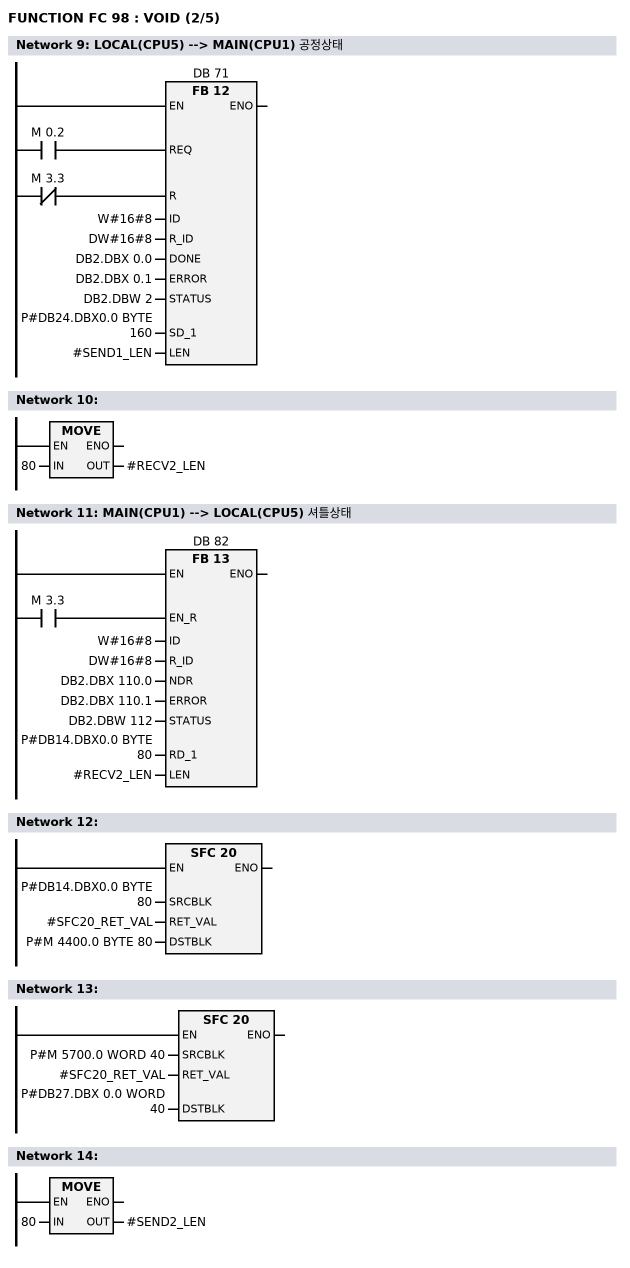

      A     M      0.2;
      =     L     14.0;
      BLD   103;
      AN    M      3.3;
      =     L     14.1;
      BLD   103;
      CALL FB    12 , DB    71 (
           REQ                      := L     14.0,
           R                        := L     14.1,
           ID                       := W#16#8,
           R_ID                     := DW#16#8,
           DONE                     := DB2.DBX    0.0,
           ERROR                    := DB2.DBX    0.1,
           STATUS                   := DB2.DBW    2,
           SD_1                     := P#DB24.DBX0.0 BYTE 160,
           LEN                      := #SEND1_LEN);
      NOP   0;
NETWORK
TITLE =

      L     80;
      T     #RECV2_LEN;
      NOP   0;
NETWORK
TITLE =MAIN(CPU1) --> LOCAL(CPU5) 셔틀상태

      A     M      3.3;
      =     L     14.0;
      BLD   103;
      CALL FB    13 , DB    82 (
           EN_R                     := L     14.0,
           ID                       := W#16#8,
           R_ID                     := DW#16#8,
           NDR                      := DB2.DBX  110.0,
           ERROR                    := DB2.DBX  110.1,
           STATUS                   := DB2.DBW  112,
           RD_1                     := P#DB14.DBX0.0 BYTE 80,
           LEN                      := #RECV2_LEN);
      NOP   0;
NETWORK
TITLE =

      CALL SFC   20 (
           SRCBLK                   := P#DB14.DBX0.0 BYTE 80,
           RET_VAL                  := #SFC20_RET_VAL,
           DSTBLK                   := P#M 4400.0 BYTE 80);
      NOP   0;
NETWORK
TITLE =

      CALL SFC   20 (
           SRCBLK                   := P#M 5700.0 WORD 40,
           RET_VAL                  := #SFC20_RET_VAL,
           DSTBLK                   := P#DB27.DBX 0.0 WORD 40);
      NOP   0;
NETWORK
TITLE =

      L     80;
      T     #SEND2_LEN;
      NOP   0;
NETWORK
TITLE =LOCAL(CPU5) --> LOCAL(CPU3) 공정상태
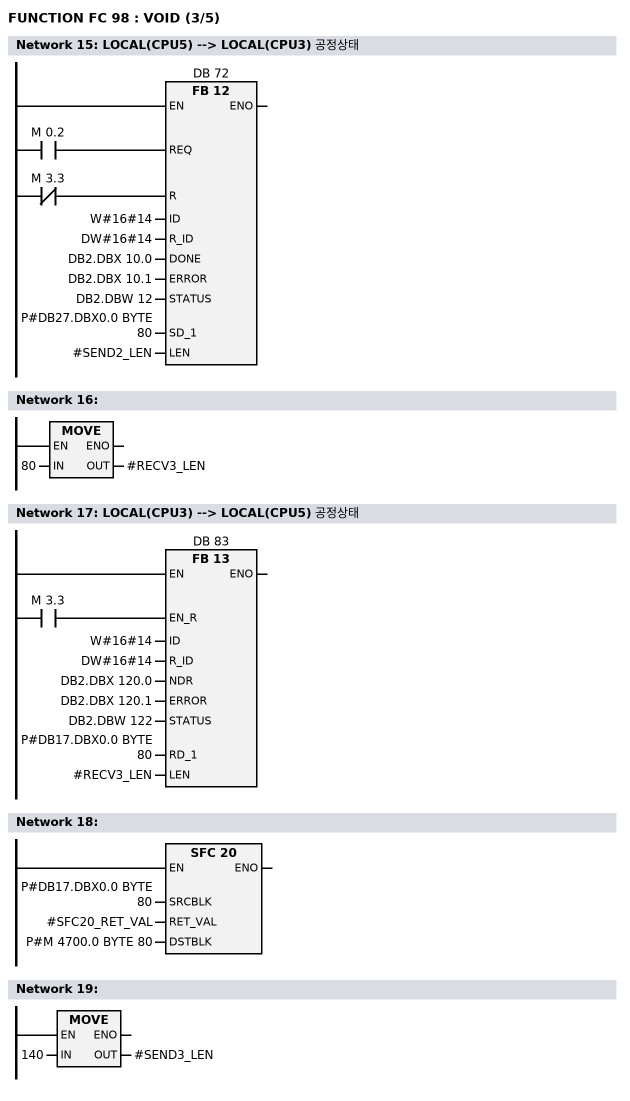

      A     M      0.2;
      =     L     14.0;
      BLD   103;
      AN    M      3.3;
      =     L     14.1;
      BLD   103;
      CALL FB    12 , DB    72 (
           REQ                      := L     14.0,
           R                        := L     14.1,
           ID                       := W#16#14,
           R_ID                     := DW#16#14,
           DONE                     := DB2.DBX   10.0,
           ERROR                    := DB2.DBX   10.1,
           STATUS                   := DB2.DBW   12,
           SD_1                     := P#DB27.DBX0.0 BYTE 80,
           LEN                      := #SEND2_LEN);
      NOP   0;
NETWORK
TITLE =

      L     80;
      T     #RECV3_LEN;
      NOP   0;
NETWORK
TITLE =LOCAL(CPU3) --> LOCAL(CPU5) 공정상태

      A     M      3.3;
      =     L     14.0;
      BLD   103;
      CALL FB    13 , DB    83 (
           EN_R                     := L     14.0,
           ID                       := W#16#14,
           R_ID                     := DW#16#14,
           NDR                      := DB2.DBX  120.0,
           ERROR                    := DB2.DBX  120.1,
           STATUS                   := DB2.DBW  122,
           RD_1                     := P#DB17.DBX0.0 BYTE 80,
           LEN                      := #RECV3_LEN);
      NOP   0;
NETWORK
TITLE =

      CALL SFC   20 (
           SRCBLK                   := P#DB17.DBX0.0 BYTE 80,
           RET_VAL                  := #SFC20_RET_VAL,
           DSTBLK                   := P#M 4700.0 BYTE 80);
      NOP   0;
NETWORK
TITLE =

      L     140;
      T     #SEND3_LEN;
      NOP   0;
NETWORK
TITLE =LOCAL(CPU5) --> MAIN(CPU1) HMI차종수정
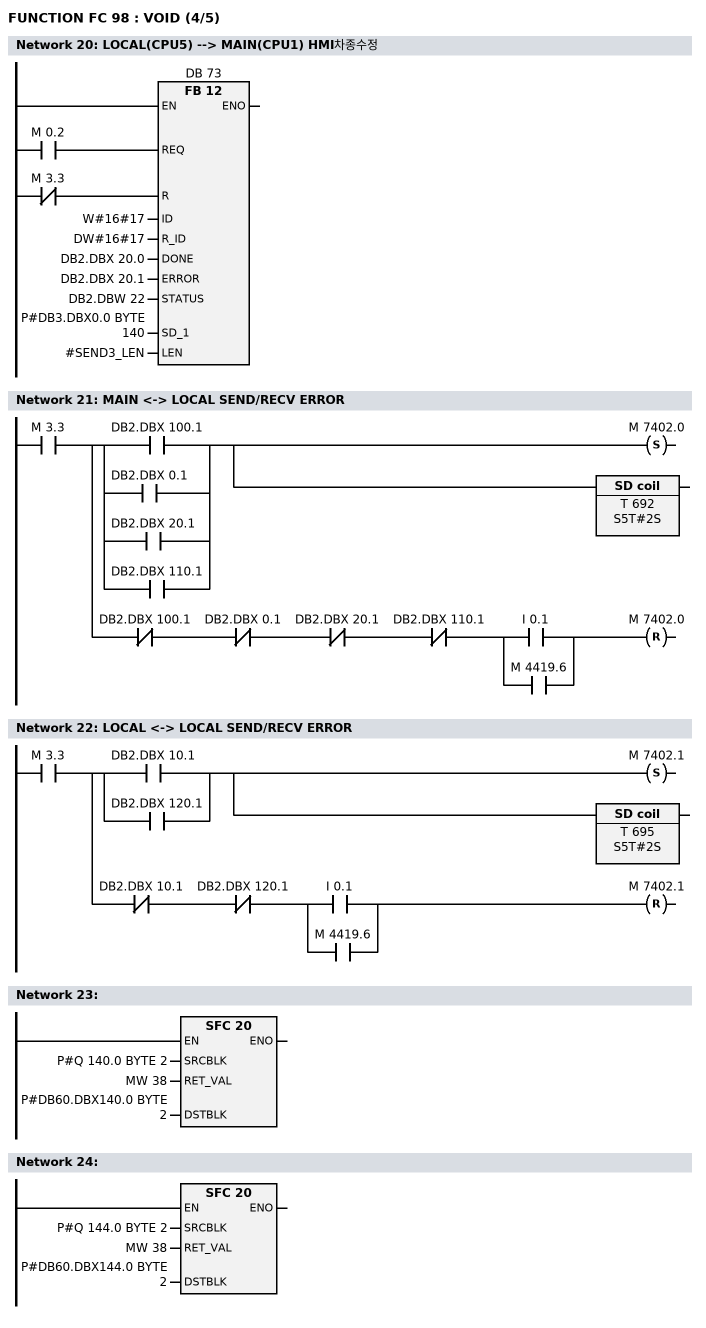

      A     M      0.2;
      =     L     14.0;
      BLD   103;
      AN    M      3.3;
      =     L     14.1;
      BLD   103;
      CALL FB    12 , DB    73 (
           REQ                      := L     14.0,
           R                        := L     14.1,
           ID                       := W#16#17,
           R_ID                     := DW#16#17,
           DONE                     := DB2.DBX   20.0,
           ERROR                    := DB2.DBX   20.1,
           STATUS                   := DB2.DBW   22,
           SD_1                     := P#DB3.DBX0.0 BYTE 140,
           LEN                      := #SEND3_LEN);
      NOP   0;
NETWORK
TITLE =MAIN <-> LOCAL SEND/RECV ERROR

      A     M      3.3;
      =     L     14.0;
      A     L     14.0;
      A(    ;
      O     DB2.DBX  100.1;
      O     DB2.DBX    0.1;
      O     DB2.DBX   20.1;
      O     DB2.DBX  110.1;
      )     ;
      S     M   7402.0;
      L     S5T#2S;
      SD    T    692;
      A     L     14.0;
      AN    DB2.DBX  100.1;
      AN    DB2.DBX    0.1;
      AN    DB2.DBX   20.1;
      AN    DB2.DBX  110.1;
      A(    ;
      O     I      0.1;
      O     M   4419.6;
      )     ;
      R     M   7402.0;
NETWORK
TITLE =LOCAL <-> LOCAL SEND/RECV ERROR

      A     M      3.3;
      =     L     14.0;
      A     L     14.0;
      A(    ;
      O     DB2.DBX   10.1;
      O     DB2.DBX  120.1;
      )     ;
      S     M   7402.1;
      L     S5T#2S;
      SD    T    695;
      A     L     14.0;
      AN    DB2.DBX   10.1;
      AN    DB2.DBX  120.1;
      A(    ;
      O     I      0.1;
      O     M   4419.6;
      )     ;
      R     M   7402.1;
NETWORK
TITLE =

      CALL SFC   20 (
           SRCBLK                   := P#Q 140.0 BYTE 2,
           RET_VAL                  := MW    38,
           DSTBLK                   := P#DB60.DBX140.0 BYTE 2);
      NOP   0;
NETWORK
TITLE =

      CALL SFC   20 (
           SRCBLK                   := P#Q 144.0 BYTE 2,
           RET_VAL                  := MW    38,
           DSTBLK                   := P#DB60.DBX144.0 BYTE 2);
      NOP   0;
NETWORK
TITLE =
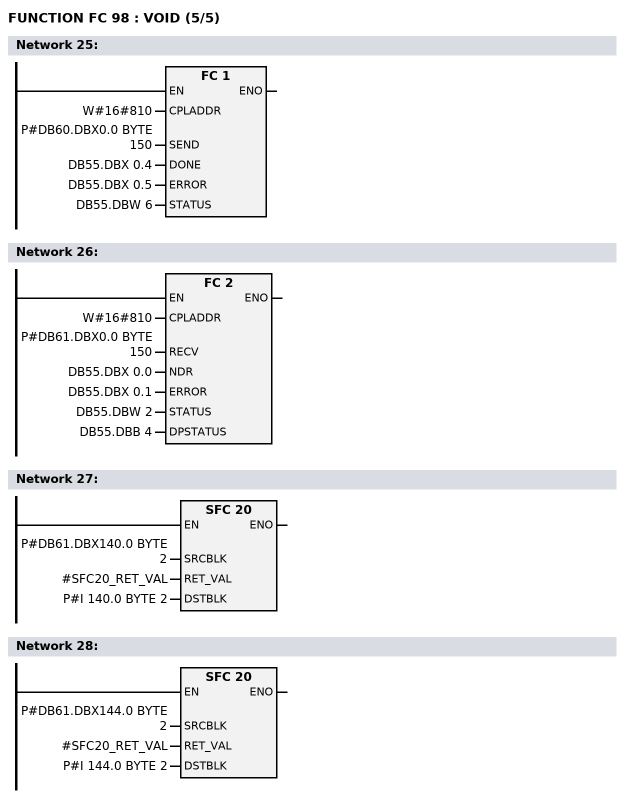

      CALL FC     1 (
           CPLADDR                  := W#16#810,
           SEND                     := P#DB60.DBX0.0 BYTE 150,
           DONE                     := DB55.DBX    0.4,
           ERROR                    := DB55.DBX    0.5,
           STATUS                   := DB55.DBW    6);
      NOP   0;
NETWORK
TITLE =

      CALL FC     2 (
           CPLADDR                  := W#16#810,
           RECV                     := P#DB61.DBX0.0 BYTE 150,
           NDR                      := DB55.DBX    0.0,
           ERROR                    := DB55.DBX    0.1,
           STATUS                   := DB55.DBW    2,
           DPSTATUS                 := DB55.DBB    4);
      NOP   0;
NETWORK
TITLE =

      CALL SFC   20 (
           SRCBLK                   := P#DB61.DBX140.0 BYTE 2,
           RET_VAL                  := #SFC20_RET_VAL,
           DSTBLK                   := P#I 140.0 BYTE 2);
      NOP   0;
NETWORK
TITLE =

      CALL SFC   20 (
           SRCBLK                   := P#DB61.DBX144.0 BYTE 2,
           RET_VAL                  := #SFC20_RET_VAL,
           DSTBLK                   := P#I 144.0 BYTE 2);
      NOP   0;
END_FUNCTION

FUNCTION FC 100 : VOID
TITLE =
VERSION : 0.1

BEGIN
NETWORK
TITLE =
